gfCNCPoint5[1220] = {X 302.7591, Y 34.0343, Z -6.3333, A 0.000, B 0.000, C 0.000 }
gfCNCPoint5[1221] = {X 293.8549, Y 34.0343, Z -6.3333, A 0.000, B 0.000, C 0.000 }
gfCNCPoint5[1222] = {X 293.8543, Y 40.9020, Z -6.3333, A 0.000, B 0.000, C 0.000 }
gfCNCPoint5[1223] = {X 294.4934, Y 41.5861, Z -6.3333, A 0.000, B 0.000, C 0.000 }
gfCNCPoint5[1224] = {X 294.9740, Y 42.3895, Z -6.3333, A 0.000, B 0.000, C 0.000 }
gfCNCPoint5[1225] = {X 295.2744, Y 43.2762, Z -6.3333, A 0.000, B 0.000, C 0.000 }
gfCNCPoint5[1226] = {X 295.3811, Y 44.2063, Z -6.3333, A 0.000, B 0.000, C 0.000 }
gfCNCPoint5[1227] = {X 295.3811, Y 45.0000, Z -6.3333, A 0.000, B 0.000, C 0.000 }
gfCNCPoint5[1228] = {X 295.2728, Y 45.9613, Z -6.3333, A 0.000, B 0.000, C 0.000 }
gfCNCPoint5[1229] = {X 294.9533, Y 46.8744, Z -6.3333, A 0.000, B 0.000, C 0.000 }
gfCNCPoint5[1230] = {X 294.4386, Y 47.6935, Z -6.3333, A 0.000, B 0.000, C 0.000 }
gfCNCPoint5[1231] = {X 293.7546, Y 48.3775, Z -6.3333, A 0.000, B 0.000, C 0.000 }
gfCNCPoint5[1232] = {X 292.9355, Y 48.8922, Z -6.3333, A 0.000, B 0.000, C 0.000 }
gfCNCPoint5[1233] = {X 292.0224, Y 49.2117, Z -6.3333, A 0.000, B 0.000, C 0.000 }
gfCNCPoint5[1234] = {X 291.0611, Y 49.3200, Z -6.3333, A 0.000, B 0.000, C 0.000 }
gfCNCPoint5[1235] = {X 284.6177, Y 49.3200, Z -6.3333, A 0.000, B 0.000, C 0.000 }
gfCNCPoint5[1236] = {X 283.6613, Y 49.2128, Z -6.3333, A 0.000, B 0.000, C 0.000 }
gfCNCPoint5[1237] = {X 282.7524, Y 48.8965, Z -6.3333, A 0.000, B 0.000, C 0.000 }
gfCNCPoint5[1238] = {X 281.9360, Y 48.3869, Z -6.3333, A 0.000, B 0.000, C 0.000 }
gfCNCPoint5[1239] = {X 281.2527, Y 47.7092, Z -6.3333, A 0.000, B 0.000, C 0.000 }
gfCNCPoint5[1240] = {X 280.7365, Y 46.8970, Z -6.3333, A 0.000, B 0.000, C 0.000 }
gfCNCPoint5[1241] = {X 280.4128, Y 45.9907, Z -6.3333, A 0.000, B 0.000, C 0.000 }
gfCNCPoint5[1242] = {X 280.2978, Y 45.0352, Z -6.3333, A 0.000, B 0.000, C 0.000 }
gfCNCPoint5[1243] = {X 280.2977, Y 44.2074, Z -6.3333, A 0.000, B 0.000, C 0.000 }
gfCNCPoint5[1244] = {X 280.4021, Y 43.2782, Z -6.3333, A 0.000, B 0.000, C 0.000 }
gfCNCPoint5[1245] = {X 280.7020, Y 42.3926, Z -6.3333, A 0.000, B 0.000, C 0.000 }
gfCNCPoint5[1246] = {X 281.1835, Y 41.5911, Z -6.3333, A 0.000, B 0.000, C 0.000 }
gfCNCPoint5[1247] = {X 281.8247, Y 40.9106, Z -6.3333, A 0.000, B 0.000, C 0.000 }
gfCNCPoint5[1248] = {X 281.8245, Y 28.5920, Z -6.3333, A 0.000, B 0.000, C 0.000 }
gfCNCPoint5[1249] = {X 277.8245, Y 28.5921, Z -6.3333, A 0.000, B 0.000, C 0.000 }
gfCNCPoint5[1250] = {X 281.9045, Y 28.5920, Z -6.3333, A 0.000, B 0.000, C 0.000 }
gfCNCPoint5[1251] = {X 281.9043, Y 16.2361, Z -6.3333, A 0.000, B 0.000, C 0.000 }
gfCNCPoint5[1252] = {X 281.2666, Y 15.5757, Z -6.3333, A 0.000, B 0.000, C 0.000 }
gfCNCPoint5[1253] = {X 280.7860, Y 14.7934, Z -6.3333, A 0.000, B 0.000, C 0.000 }
gfCNCPoint5[1254] = {X 280.4850, Y 13.9261, Z -6.3333, A 0.000, B 0.000, C 0.000 }
gfCNCPoint5[1255] = {X 280.3778, Y 13.0143, Z -6.3333, A 0.000, B 0.000, C 0.000 }
gfCNCPoint5[1256] = {X 280.3777, Y 12.1868, Z -6.3333, A 0.000, B 0.000, C 0.000 }
gfCNCPoint5[1257] = {X 280.4840, Y 11.2433, Z -6.3333, A 0.000, B 0.000, C 0.000 }
gfCNCPoint5[1258] = {X 280.7976, Y 10.3472, Z -6.3333, A 0.000, B 0.000, C 0.000 }
gfCNCPoint5[1259] = {X 281.3027, Y 9.5432, Z -6.3333, A 0.000, B 0.000, C 0.000 }
gfCNCPoint5[1260] = {X 281.9741, Y 8.8719, Z -6.3333, A 0.000, B 0.000, C 0.000 }
gfCNCPoint5[1261] = {X 282.7780, Y 8.3667, Z -6.3333, A 0.000, B 0.000, C 0.000 }
gfCNCPoint5[1262] = {X 283.6742, Y 8.0531, Z -6.3333, A 0.000, B 0.000, C 0.000 }
gfCNCPoint5[1263] = {X 284.6177, Y 7.9468, Z -6.3333, A 0.000, B 0.000, C 0.000 }
gfCNCPoint5[1264] = {X 291.0611, Y 7.9468, Z -6.3333, A 0.000, B 0.000, C 0.000 }
gfCNCPoint5[1265] = {X 292.0046, Y 8.0531, Z -6.3333, A 0.000, B 0.000, C 0.000 }
gfCNCPoint5[1266] = {X 292.9008, Y 8.3667, Z -6.3333, A 0.000, B 0.000, C 0.000 }
gfCNCPoint5[1267] = {X 293.7047, Y 8.8718, Z -6.3333, A 0.000, B 0.000, C 0.000 }
gfCNCPoint5[1268] = {X 294.3761, Y 9.5432, Z -6.3333, A 0.000, B 0.000, C 0.000 }
gfCNCPoint5[1269] = {X 294.8812, Y 10.3471, Z -6.3333, A 0.000, B 0.000, C 0.000 }
gfCNCPoint5[1270] = {X 295.1948, Y 11.2433, Z -6.3333, A 0.000, B 0.000, C 0.000 }
gfCNCPoint5[1271] = {X 295.3011, Y 12.1868, Z -6.3333, A 0.000, B 0.000, C 0.000 }
gfCNCPoint5[1272] = {X 295.3011, Y 12.9782, Z -6.3333, A 0.000, B 0.000, C 0.000 }
gfCNCPoint5[1273] = {X 295.1997, Y 13.8997, Z -6.3333, A 0.000, B 0.000, C 0.000 }
gfCNCPoint5[1274] = {X 294.9003, Y 14.7771, Z -6.3333, A 0.000, B 0.000, C 0.000 }
gfCNCPoint5[1275] = {X 294.4175, Y 15.5685, Z -6.3333, A 0.000, B 0.000, C 0.000 }
gfCNCPoint5[1276] = {X 293.7742, Y 16.2360, Z -6.3333, A 0.000, B 0.000, C 0.000 }
gfCNCPoint5[1277] = {X 293.7752, Y 22.2765, Z -6.3333, A 0.000, B 0.000, C 0.000 }
gfCNCPoint5[1278] = {X 302.8386, Y 22.2765, Z -6.3333, A 0.000, B 0.000, C 0.000 }
gfCNCPoint5[1279] = {X 302.8437, Y 16.2401, Z -6.3333, A 0.000, B 0.000, C 0.000 }
gfCNCPoint5[1280] = {X 302.2043, Y 15.5797, Z -6.3333, A 0.000, B 0.000, C 0.000 }
gfCNCPoint5[1281] = {X 301.7222, Y 14.7970, Z -6.3333, A 0.000, B 0.000, C 0.000 }
gfCNCPoint5[1282] = {X 301.4202, Y 13.9287, Z -6.3333, A 0.000, B 0.000, C 0.000 }
gfCNCPoint5[1283] = {X 301.3124, Y 13.0158, Z -6.3333, A 0.000, B 0.000, C 0.000 }
gfCNCPoint5[1284] = {X 301.3123, Y 12.1868, Z -6.3333, A 0.000, B 0.000, C 0.000 }
gfCNCPoint5[1285] = {X 301.4186, Y 11.2433, Z -6.3333, A 0.000, B 0.000, C 0.000 }
gfCNCPoint5[1286] = {X 301.7321, Y 10.3471, Z -6.3333, A 0.000, B 0.000, C 0.000 }
gfCNCPoint5[1287] = {X 302.2373, Y 9.5432, Z -6.3333, A 0.000, B 0.000, C 0.000 }
gfCNCPoint5[1288] = {X 302.9087, Y 8.8718, Z -6.3333, A 0.000, B 0.000, C 0.000 }
gfCNCPoint5[1289] = {X 303.7126, Y 8.3667, Z -6.3333, A 0.000, B 0.000, C 0.000 }
gfCNCPoint5[1290] = {X 304.6088, Y 8.0531, Z -6.3333, A 0.000, B 0.000, C 0.000 }
gfCNCPoint5[1291] = {X 305.5523, Y 7.9468, Z -6.3333, A 0.000, B 0.000, C 0.000 }
gfCNCPoint5[1292] = {X 311.9957, Y 7.9468, Z -6.3333, A 0.000, B 0.000, C 0.000 }
gfCNCPoint5[1293] = {X 312.9392, Y 8.0531, Z -6.3333, A 0.000, B 0.000, C 0.000 }
gfCNCPoint5[1294] = {X 313.8354, Y 8.3667, Z -6.3333, A 0.000, B 0.000, C 0.000 }
gfCNCPoint5[1295] = {X 314.6393, Y 8.8718, Z -6.3333, A 0.000, B 0.000, C 0.000 }
gfCNCPoint5[1296] = {X 315.3107, Y 9.5432, Z -6.3333, A 0.000, B 0.000, C 0.000 }
gfCNCPoint5[1297] = {X 315.8158, Y 10.3471, Z -6.3333, A 0.000, B 0.000, C 0.000 }
gfCNCPoint5[1298] = {X 316.1294, Y 11.2433, Z -6.3333, A 0.000, B 0.000, C 0.000 }
gfCNCPoint5[1299] = {X 316.2357, Y 12.1868, Z -6.3333, A 0.000, B 0.000, C 0.000 }
gfCNCPoint5[1300] = {X 316.2357, Y 12.9782, Z -6.3333, A 0.000, B 0.000, C 0.000 }
gfCNCPoint5[1301] = {X 316.1344, Y 13.8995, Z -6.3333, A 0.000, B 0.000, C 0.000 }
gfCNCPoint5[1302] = {X 315.8352, Y 14.7768, Z -6.3333, A 0.000, B 0.000, C 0.000 }
gfCNCPoint5[1303] = {X 315.3526, Y 15.5682, Z -6.3333, A 0.000, B 0.000, C 0.000 }
gfCNCPoint5[1304] = {X 314.7095, Y 16.2358, Z -6.3333, A 0.000, B 0.000, C 0.000 }
gfCNCPoint5[1305] = {X 314.7087, Y 40.9513, Z -6.3333, A 0.000, B 0.000, C 0.000 }
gfCNCPoint5[1306] = {X 314.7370, Y 40.9741, Z -6.3333, A 0.000, B 0.000, C 0.000 }
gfCNCPoint5[1307] = {X 315.3634, Y 41.6327, Z -6.3333, A 0.000, B 0.000, C 0.000 }
gfCNCPoint5[1308] = {X 315.8351, Y 42.4096, Z -6.3333, A 0.000, B 0.000, C 0.000 }
gfCNCPoint5[1309] = {X 316.1303, Y 43.2692, Z -6.3333, A 0.000, B 0.000, C 0.000 }
gfCNCPoint5[1310] = {X 316.2356, Y 44.1720, Z -6.3333, A 0.000, B 0.000, C 0.000 }
gfCNCPoint5[1311] = {X 316.2357, Y 45.0000, Z -6.3333, A 0.000, B 0.000, C 0.000 }
gfCNCPoint5[1312] = {X 316.1294, Y 45.9435, Z -6.3333, A 0.000, B 0.000, C 0.000 }
gfCNCPoint5[1313] = {X 315.8158, Y 46.8397, Z -6.3333, A 0.000, B 0.000, C 0.000 }
gfCNCPoint5[1314] = {X 315.3107, Y 47.6436, Z -6.3333, A 0.000, B 0.000, C 0.000 }
gfCNCPoint5[1315] = {X 314.6393, Y 48.3150, Z -6.3333, A 0.000, B 0.000, C 0.000 }
gfCNCPoint5[1316] = {X 313.8354, Y 48.8201, Z -6.3333, A 0.000, B 0.000, C 0.000 }
gfCNCPoint5[1317] = {X 312.9392, Y 49.1337, Z -6.3333, A 0.000, B 0.000, C 0.000 }
gfCNCPoint5[1318] = {X 311.9957, Y 49.2400, Z -6.3333, A 0.000, B 0.000, C 0.000 }
gfCNCPoint5[1319] = {X 305.5523, Y 49.2400, Z -6.3333, A 0.000, B 0.000, C 0.000 }
gfCNCPoint5[1320] = {X 304.6135, Y 49.1348, Z -6.3333, A 0.000, B 0.000, C 0.000 }
gfCNCPoint5[1321] = {X 303.7214, Y 48.8243, Z -6.3333, A 0.000, B 0.000, C 0.000 }
gfCNCPoint5[1322] = {X 302.9201, Y 48.3241, Z -6.3333, A 0.000, B 0.000, C 0.000 }
gfCNCPoint5[1323] = {X 302.2495, Y 47.6588, Z -6.3333, A 0.000, B 0.000, C 0.000 }
gfCNCPoint5[1324] = {X 301.7428, Y 46.8616, Z -6.3333, A 0.000, B 0.000, C 0.000 }
gfCNCPoint5[1325] = {X 301.4252, Y 45.9720, Z -6.3333, A 0.000, B 0.000, C 0.000 }
gfCNCPoint5[1326] = {X 301.3124, Y 45.0341, Z -6.3333, A 0.000, B 0.000, C 0.000 }
gfCNCPoint5[1327] = {X 301.3123, Y 44.2032, Z -6.3333, A 0.000, B 0.000, C 0.000 }
gfCNCPoint5[1328] = {X 301.4296, Y 43.2746, Z -6.3333, A 0.000, B 0.000, C 0.000 }
gfCNCPoint5[1329] = {X 301.7327, Y 42.3890, Z -6.3333, A 0.000, B 0.000, C 0.000 }
gfCNCPoint5[1330] = {X 302.2091, Y 41.5833, Z -6.3333, A 0.000, B 0.000, C 0.000 }
gfCNCPoint5[1331] = {X 302.8391, Y 40.8909, Z -6.3333, A 0.000, B 0.000, C 0.000 }
gfCNCPoint5[1332] = {X 302.8391, Y 33.9543, Z -6.3333, A 0.000, B 0.000, C 0.000 }
gfCNCPoint5[1333] = {X 293.7749, Y 33.9543, Z -6.3333, A 0.000, B 0.000, C 0.000 }
gfCNCPoint5[1334] = {X 293.7743, Y 40.9388, Z -6.3333, A 0.000, B 0.000, C 0.000 }
gfCNCPoint5[1335] = {X 294.4130, Y 41.6124, Z -6.3333, A 0.000, B 0.000, C 0.000 }
gfCNCPoint5[1336] = {X 294.8937, Y 42.4065, Z -6.3333, A 0.000, B 0.000, C 0.000 }
gfCNCPoint5[1337] = {X 295.1944, Y 43.2848, Z -6.3333, A 0.000, B 0.000, C 0.000 }
gfCNCPoint5[1338] = {X 295.3011, Y 44.2069, Z -6.3333, A 0.000, B 0.000, C 0.000 }
gfCNCPoint5[1339] = {X 295.3011, Y 45.0000, Z -6.3333, A 0.000, B 0.000, C 0.000 }
gfCNCPoint5[1340] = {X 295.1948, Y 45.9435, Z -6.3333, A 0.000, B 0.000, C 0.000 }
gfCNCPoint5[1341] = {X 294.8812, Y 46.8397, Z -6.3333, A 0.000, B 0.000, C 0.000 }
gfCNCPoint5[1342] = {X 294.3761, Y 47.6436, Z -6.3333, A 0.000, B 0.000, C 0.000 }
gfCNCPoint5[1343] = {X 293.7047, Y 48.3150, Z -6.3333, A 0.000, B 0.000, C 0.000 }
gfCNCPoint5[1344] = {X 292.9008, Y 48.8201, Z -6.3333, A 0.000, B 0.000, C 0.000 }
gfCNCPoint5[1345] = {X 292.0046, Y 49.1337, Z -6.3333, A 0.000, B 0.000, C 0.000 }
gfCNCPoint5[1346] = {X 291.0611, Y 49.2400, Z -6.3333, A 0.000, B 0.000, C 0.000 }
gfCNCPoint5[1347] = {X 284.6177, Y 49.2400, Z -6.3333, A 0.000, B 0.000, C 0.000 }
gfCNCPoint5[1348] = {X 283.6790, Y 49.1348, Z -6.3333, A 0.000, B 0.000, C 0.000 }
gfCNCPoint5[1349] = {X 282.7869, Y 48.8244, Z -6.3333, A 0.000, B 0.000, C 0.000 }
gfCNCPoint5[1350] = {X 281.9857, Y 48.3242, Z -6.3333, A 0.000, B 0.000, C 0.000 }
gfCNCPoint5[1351] = {X 281.3150, Y 47.6590, Z -6.3333, A 0.000, B 0.000, C 0.000 }
gfCNCPoint5[1352] = {X 280.8083, Y 46.8619, Z -6.3333, A 0.000, B 0.000, C 0.000 }
gfCNCPoint5[1353] = {X 280.4907, Y 45.9723, Z -6.3333, A 0.000, B 0.000, C 0.000 }
gfCNCPoint5[1354] = {X 280.3778, Y 45.0345, Z -6.3333, A 0.000, B 0.000, C 0.000 }
gfCNCPoint5[1355] = {X 280.3777, Y 44.2077, Z -6.3333, A 0.000, B 0.000, C 0.000 }
gfCNCPoint5[1356] = {X 280.4822, Y 43.2867, Z -6.3333, A 0.000, B 0.000, C 0.000 }
gfCNCPoint5[1357] = {X 280.7823, Y 42.4096, Z -6.3333, A 0.000, B 0.000, C 0.000 }
gfCNCPoint5[1358] = {X 281.2640, Y 41.6176, Z -6.3333, A 0.000, B 0.000, C 0.000 }
gfCNCPoint5[1359] = {X 281.9047, Y 40.9476, Z -6.3333, A 0.000, B 0.000, C 0.000 }
gfCNCPoint5[1360] = {X 281.9045, Y 28.5920, Z -6.3333, A 0.000, B 0.000, C 0.000 }
gfCNCPoint5[1361] = {X 277.9045, Y 28.5921, Z -6.3333, A 0.000, B 0.000, C 0.000 }
gfCNCPoint5[1362] = {X 281.9845, Y 28.5920, Z -6.3333, A 0.000, B 0.000, C 0.000 }
gfCNCPoint5[1363] = {X 281.9843, Y 16.1984, Z -6.3333, A 0.000, B 0.000, C 0.000 }
gfCNCPoint5[1364] = {X 281.3470, Y 15.5487, Z -6.3333, A 0.000, B 0.000, C 0.000 }
gfCNCPoint5[1365] = {X 280.8663, Y 14.7760, Z -6.3333, A 0.000, B 0.000, C 0.000 }
gfCNCPoint5[1366] = {X 280.5651, Y 13.9173, Z -6.3333, A 0.000, B 0.000, C 0.000 }
gfCNCPoint5[1367] = {X 280.4578, Y 13.0136, Z -6.3333, A 0.000, B 0.000, C 0.000 }
gfCNCPoint5[1368] = {X 280.4577, Y 12.1868, Z -6.3333, A 0.000, B 0.000, C 0.000 }
gfCNCPoint5[1369] = {X 280.5620, Y 11.2611, Z -6.3333, A 0.000, B 0.000, C 0.000 }
gfCNCPoint5[1370] = {X 280.8696, Y 10.3819, Z -6.3333, A 0.000, B 0.000, C 0.000 }
gfCNCPoint5[1371] = {X 281.3652, Y 9.5931, Z -6.3333, A 0.000, B 0.000, C 0.000 }
gfCNCPoint5[1372] = {X 282.0240, Y 8.9344, Z -6.3333, A 0.000, B 0.000, C 0.000 }
gfCNCPoint5[1373] = {X 282.8127, Y 8.4388, Z -6.3333, A 0.000, B 0.000, C 0.000 }
gfCNCPoint5[1374] = {X 283.6920, Y 8.1311, Z -6.3333, A 0.000, B 0.000, C 0.000 }
gfCNCPoint5[1375] = {X 284.6177, Y 8.0268, Z -6.3333, A 0.000, B 0.000, C 0.000 }
gfCNCPoint5[1376] = {X 291.0611, Y 8.0268, Z -6.3333, A 0.000, B 0.000, C 0.000 }
gfCNCPoint5[1377] = {X 291.9868, Y 8.1311, Z -6.3333, A 0.000, B 0.000, C 0.000 }
gfCNCPoint5[1378] = {X 292.8661, Y 8.4388, Z -6.3333, A 0.000, B 0.000, C 0.000 }
gfCNCPoint5[1379] = {X 293.6549, Y 8.9344, Z -6.3333, A 0.000, B 0.000, C 0.000 }
gfCNCPoint5[1380] = {X 294.3136, Y 9.5931, Z -6.3333, A 0.000, B 0.000, C 0.000 }
gfCNCPoint5[1381] = {X 294.8092, Y 10.3819, Z -6.3333, A 0.000, B 0.000, C 0.000 }
gfCNCPoint5[1382] = {X 295.1168, Y 11.2611, Z -6.3333, A 0.000, B 0.000, C 0.000 }
gfCNCPoint5[1383] = {X 295.2211, Y 12.1868, Z -6.3333, A 0.000, B 0.000, C 0.000 }
gfCNCPoint5[1384] = {X 295.2211, Y 12.9782, Z -6.3333, A 0.000, B 0.000, C 0.000 }
gfCNCPoint5[1385] = {X 295.1255, Y 13.8649, Z -6.3333, A 0.000, B 0.000, C 0.000 }
gfCNCPoint5[1386] = {X 294.8430, Y 14.7110, Z -6.3333, A 0.000, B 0.000, C 0.000 }
gfCNCPoint5[1387] = {X 294.3867, Y 15.4773, Z -6.3333, A 0.000, B 0.000, C 0.000 }
gfCNCPoint5[1388] = {X 293.7775, Y 16.1288, Z -6.3333, A 0.000, B 0.000, C 0.000 }
gfCNCPoint5[1389] = {X 293.6942, Y 16.1987, Z -6.3333, A 0.000, B 0.000, C 0.000 }
gfCNCPoint5[1390] = {X 293.6952, Y 22.3565, Z -6.3333, A 0.000, B 0.000, C 0.000 }
gfCNCPoint5[1391] = {X 302.9185, Y 22.3565, Z -6.3333, A 0.000, B 0.000, C 0.000 }
gfCNCPoint5[1392] = {X 302.9237, Y 16.2024, Z -6.3333, A 0.000, B 0.000, C 0.000 }
gfCNCPoint5[1393] = {X 302.2848, Y 15.5527, Z -6.3333, A 0.000, B 0.000, C 0.000 }
gfCNCPoint5[1394] = {X 301.8026, Y 14.7796, Z -6.3333, A 0.000, B 0.000, C 0.000 }
gfCNCPoint5[1395] = {X 301.5003, Y 13.9199, Z -6.3333, A 0.000, B 0.000, C 0.000 }
gfCNCPoint5[1396] = {X 301.3924, Y 13.0151, Z -6.3333, A 0.000, B 0.000, C 0.000 }
gfCNCPoint5[1397] = {X 301.3923, Y 12.1868, Z -6.3333, A 0.000, B 0.000, C 0.000 }
gfCNCPoint5[1398] = {X 301.4966, Y 11.2611, Z -6.3333, A 0.000, B 0.000, C 0.000 }
gfCNCPoint5[1399] = {X 301.8042, Y 10.3819, Z -6.3333, A 0.000, B 0.000, C 0.000 }
gfCNCPoint5[1400] = {X 302.2998, Y 9.5931, Z -6.3333, A 0.000, B 0.000, C 0.000 }
gfCNCPoint5[1401] = {X 302.9585, Y 8.9344, Z -6.3333, A 0.000, B 0.000, C 0.000 }
gfCNCPoint5[1402] = {X 303.7473, Y 8.4388, Z -6.3333, A 0.000, B 0.000, C 0.000 }
gfCNCPoint5[1403] = {X 304.6266, Y 8.1311, Z -6.3333, A 0.000, B 0.000, C 0.000 }
gfCNCPoint5[1404] = {X 305.5523, Y 8.0268, Z -6.3333, A 0.000, B 0.000, C 0.000 }
gfCNCPoint5[1405] = {X 311.9957, Y 8.0268, Z -6.3333, A 0.000, B 0.000, C 0.000 }
gfCNCPoint5[1406] = {X 312.9214, Y 8.1311, Z -6.3333, A 0.000, B 0.000, C 0.000 }
gfCNCPoint5[1407] = {X 313.8007, Y 8.4388, Z -6.3333, A 0.000, B 0.000, C 0.000 }
gfCNCPoint5[1408] = {X 314.5894, Y 8.9344, Z -6.3333, A 0.000, B 0.000, C 0.000 }
gfCNCPoint5[1409] = {X 315.2481, Y 9.5931, Z -6.3333, A 0.000, B 0.000, C 0.000 }
gfCNCPoint5[1410] = {X 315.7438, Y 10.3819, Z -6.3333, A 0.000, B 0.000, C 0.000 }
gfCNCPoint5[1411] = {X 316.0514, Y 11.2611, Z -6.3333, A 0.000, B 0.000, C 0.000 }
gfCNCPoint5[1412] = {X 316.1557, Y 12.1868, Z -6.3333, A 0.000, B 0.000, C 0.000 }
gfCNCPoint5[1413] = {X 316.1557, Y 12.9782, Z -6.3333, A 0.000, B 0.000, C 0.000 }
gfCNCPoint5[1414] = {X 316.0542, Y 13.8913, Z -6.3333, A 0.000, B 0.000, C 0.000 }
gfCNCPoint5[1415] = {X 315.7548, Y 14.7598, Z -6.3333, A 0.000, B 0.000, C 0.000 }
gfCNCPoint5[1416] = {X 315.2721, Y 15.5414, Z -6.3333, A 0.000, B 0.000, C 0.000 }
gfCNCPoint5[1417] = {X 314.6295, Y 16.1981, Z -6.3333, A 0.000, B 0.000, C 0.000 }
gfCNCPoint5[1418] = {X 314.6287, Y 40.9896, Z -6.3333, A 0.000, B 0.000, C 0.000 }
gfCNCPoint5[1419] = {X 314.6838, Y 41.0339, Z -6.3333, A 0.000, B 0.000, C 0.000 }
gfCNCPoint5[1420] = {X 315.2990, Y 41.6801, Z -6.3333, A 0.000, B 0.000, C 0.000 }
gfCNCPoint5[1421] = {X 315.7622, Y 42.4427, Z -6.3333, A 0.000, B 0.000, C 0.000 }
gfCNCPoint5[1422] = {X 316.0522, Y 43.2864, Z -6.3333, A 0.000, B 0.000, C 0.000 }
gfCNCPoint5[1423] = {X 316.1556, Y 44.1727, Z -6.3333, A 0.000, B 0.000, C 0.000 }
gfCNCPoint5[1424] = {X 316.1557, Y 45.0000, Z -6.3333, A 0.000, B 0.000, C 0.000 }
gfCNCPoint5[1425] = {X 316.0514, Y 45.9257, Z -6.3333, A 0.000, B 0.000, C 0.000 }
gfCNCPoint5[1426] = {X 315.7438, Y 46.8050, Z -6.3333, A 0.000, B 0.000, C 0.000 }
gfCNCPoint5[1427] = {X 315.2481, Y 47.5937, Z -6.3333, A 0.000, B 0.000, C 0.000 }
gfCNCPoint5[1428] = {X 314.5894, Y 48.2524, Z -6.3333, A 0.000, B 0.000, C 0.000 }
gfCNCPoint5[1429] = {X 313.8007, Y 48.7480, Z -6.3333, A 0.000, B 0.000, C 0.000 }
gfCNCPoint5[1430] = {X 312.9214, Y 49.0557, Z -6.3333, A 0.000, B 0.000, C 0.000 }
gfCNCPoint5[1431] = {X 311.9957, Y 49.1600, Z -6.3333, A 0.000, B 0.000, C 0.000 }
gfCNCPoint5[1432] = {X 305.5523, Y 49.1600, Z -6.3333, A 0.000, B 0.000, C 0.000 }
gfCNCPoint5[1433] = {X 304.6312, Y 49.0568, Z -6.3333, A 0.000, B 0.000, C 0.000 }
gfCNCPoint5[1434] = {X 303.7559, Y 48.7522, Z -6.3333, A 0.000, B 0.000, C 0.000 }
gfCNCPoint5[1435] = {X 302.9698, Y 48.2613, Z -6.3333, A 0.000, B 0.000, C 0.000 }
gfCNCPoint5[1436] = {X 302.3118, Y 47.6087, Z -6.3333, A 0.000, B 0.000, C 0.000 }
gfCNCPoint5[1437] = {X 301.8147, Y 46.8265, Z -6.3333, A 0.000, B 0.000, C 0.000 }
gfCNCPoint5[1438] = {X 301.5030, Y 45.9537, Z -6.3333, A 0.000, B 0.000, C 0.000 }
gfCNCPoint5[1439] = {X 301.3924, Y 45.0335, Z -6.3333, A 0.000, B 0.000, C 0.000 }
gfCNCPoint5[1440] = {X 301.3923, Y 44.2051, Z -6.3333, A 0.000, B 0.000, C 0.000 }
gfCNCPoint5[1441] = {X 301.5095, Y 43.2839, Z -6.3333, A 0.000, B 0.000, C 0.000 }
gfCNCPoint5[1442] = {X 301.8128, Y 42.4063, Z -6.3333, A 0.000, B 0.000, C 0.000 }
gfCNCPoint5[1443] = {X 302.2894, Y 41.6093, Z -6.3333, A 0.000, B 0.000, C 0.000 }
gfCNCPoint5[1444] = {X 302.9191, Y 40.9268, Z -6.3333, A 0.000, B 0.000, C 0.000 }
gfCNCPoint5[1445] = {X 302.9191, Y 33.8743, Z -6.3333, A 0.000, B 0.000, C 0.000 }
gfCNCPoint5[1446] = {X 293.6950, Y 33.8743, Z -6.3333, A 0.000, B 0.000, C 0.000 }
gfCNCPoint5[1447] = {X 293.6943, Y 40.9760, Z -6.3333, A 0.000, B 0.000, C 0.000 }
gfCNCPoint5[1448] = {X 294.3326, Y 41.6390, Z -6.3333, A 0.000, B 0.000, C 0.000 }
gfCNCPoint5[1449] = {X 294.8134, Y 42.4237, Z -6.3333, A 0.000, B 0.000, C 0.000 }
gfCNCPoint5[1450] = {X 295.1143, Y 43.2935, Z -6.3333, A 0.000, B 0.000, C 0.000 }
gfCNCPoint5[1451] = {X 295.2211, Y 44.2076, Z -6.3333, A 0.000, B 0.000, C 0.000 }
gfCNCPoint5[1452] = {X 295.2211, Y 45.0000, Z -6.3333, A 0.000, B 0.000, C 0.000 }
gfCNCPoint5[1453] = {X 295.1168, Y 45.9257, Z -6.3333, A 0.000, B 0.000, C 0.000 }
gfCNCPoint5[1454] = {X 294.8092, Y 46.8050, Z -6.3333, A 0.000, B 0.000, C 0.000 }
gfCNCPoint5[1455] = {X 294.3136, Y 47.5937, Z -6.3333, A 0.000, B 0.000, C 0.000 }
gfCNCPoint5[1456] = {X 293.6549, Y 48.2524, Z -6.3333, A 0.000, B 0.000, C 0.000 }
gfCNCPoint5[1457] = {X 292.8661, Y 48.7480, Z -6.3333, A 0.000, B 0.000, C 0.000 }
gfCNCPoint5[1458] = {X 291.9868, Y 49.0557, Z -6.3333, A 0.000, B 0.000, C 0.000 }
gfCNCPoint5[1459] = {X 291.0611, Y 49.1600, Z -6.3333, A 0.000, B 0.000, C 0.000 }
gfCNCPoint5[1460] = {X 284.6177, Y 49.1600, Z -6.3333, A 0.000, B 0.000, C 0.000 }
gfCNCPoint5[1461] = {X 283.6967, Y 49.0568, Z -6.3333, A 0.000, B 0.000, C 0.000 }
gfCNCPoint5[1462] = {X 282.8214, Y 48.7522, Z -6.3333, A 0.000, B 0.000, C 0.000 }
gfCNCPoint5[1463] = {X 282.0353, Y 48.2615, Z -6.3333, A 0.000, B 0.000, C 0.000 }
gfCNCPoint5[1464] = {X 281.3774, Y 47.6088, Z -6.3333, A 0.000, B 0.000, C 0.000 }
gfCNCPoint5[1465] = {X 280.8802, Y 46.8267, Z -6.3333, A 0.000, B 0.000, C 0.000 }
gfCNCPoint5[1466] = {X 280.5685, Y 45.9540, Z -6.3333, A 0.000, B 0.000, C 0.000 }
gfCNCPoint5[1467] = {X 280.4578, Y 45.0339, Z -6.3333, A 0.000, B 0.000, C 0.000 }
gfCNCPoint5[1468] = {X 280.4577, Y 44.2081, Z -6.3333, A 0.000, B 0.000, C 0.000 }
gfCNCPoint5[1469] = {X 280.5623, Y 43.2952, Z -6.3333, A 0.000, B 0.000, C 0.000 }
gfCNCPoint5[1470] = {X 280.8627, Y 42.4267, Z -6.3333, A 0.000, B 0.000, C 0.000 }
gfCNCPoint5[1471] = {X 281.3445, Y 41.6443, Z -6.3333, A 0.000, B 0.000, C 0.000 }
gfCNCPoint5[1472] = {X 281.9847, Y 40.9851, Z -6.3333, A 0.000, B 0.000, C 0.000 }
gfCNCPoint5[1473] = {X 281.9845, Y 28.5920, Z -6.3333, A 0.000, B 0.000, C 0.000 }
gfCNCPoint5[1474] = {X 277.9845, Y 28.5921, Z -6.3333, A 0.000, B 0.000, C 0.000 }
gfCNCPoint5[1475] = {X 282.0645, Y 28.5920, Z -6.3333, A 0.000, B 0.000, C 0.000 }
gfCNCPoint5[1476] = {X 282.0643, Y 16.1603, Z -6.3333, A 0.000, B 0.000, C 0.000 }
gfCNCPoint5[1477] = {X 281.4275, Y 15.5215, Z -6.3333, A 0.000, B 0.000, C 0.000 }
gfCNCPoint5[1478] = {X 280.9467, Y 14.7585, Z -6.3333, A 0.000, B 0.000, C 0.000 }
gfCNCPoint5[1479] = {X 280.6452, Y 13.9084, Z -6.3333, A 0.000, B 0.000, C 0.000 }
gfCNCPoint5[1480] = {X 280.5378, Y 13.0129, Z -6.3333, A 0.000, B 0.000, C 0.000 }
gfCNCPoint5[1481] = {X 280.5377, Y 12.1868, Z -6.3333, A 0.000, B 0.000, C 0.000 }
gfCNCPoint5[1482] = {X 280.6400, Y 11.2789, Z -6.3333, A 0.000, B 0.000, C 0.000 }
gfCNCPoint5[1483] = {X 280.9417, Y 10.4166, Z -6.3333, A 0.000, B 0.000, C 0.000 }
gfCNCPoint5[1484] = {X 281.4278, Y 9.6430, Z -6.3333, A 0.000, B 0.000, C 0.000 }
gfCNCPoint5[1485] = {X 282.0738, Y 8.9969, Z -6.3333, A 0.000, B 0.000, C 0.000 }
gfCNCPoint5[1486] = {X 282.8474, Y 8.5109, Z -6.3333, A 0.000, B 0.000, C 0.000 }
gfCNCPoint5[1487] = {X 283.7098, Y 8.2091, Z -6.3333, A 0.000, B 0.000, C 0.000 }
gfCNCPoint5[1488] = {X 284.6177, Y 8.1068, Z -6.3333, A 0.000, B 0.000, C 0.000 }
gfCNCPoint5[1489] = {X 291.0611, Y 8.1068, Z -6.3333, A 0.000, B 0.000, C 0.000 }
gfCNCPoint5[1490] = {X 291.9690, Y 8.2091, Z -6.3333, A 0.000, B 0.000, C 0.000 }
gfCNCPoint5[1491] = {X 292.8314, Y 8.5109, Z -6.3333, A 0.000, B 0.000, C 0.000 }
gfCNCPoint5[1492] = {X 293.6050, Y 8.9969, Z -6.3333, A 0.000, B 0.000, C 0.000 }
gfCNCPoint5[1493] = {X 294.2510, Y 9.6430, Z -6.3333, A 0.000, B 0.000, C 0.000 }
gfCNCPoint5[1494] = {X 294.7371, Y 10.4166, Z -6.3333, A 0.000, B 0.000, C 0.000 }
gfCNCPoint5[1495] = {X 295.0388, Y 11.2789, Z -6.3333, A 0.000, B 0.000, C 0.000 }
gfCNCPoint5[1496] = {X 295.1411, Y 12.1868, Z -6.3333, A 0.000, B 0.000, C 0.000 }
gfCNCPoint5[1497] = {X 295.1411, Y 12.9782, Z -6.3333, A 0.000, B 0.000, C 0.000 }
gfCNCPoint5[1498] = {X 295.0473, Y 13.8479, Z -6.3333, A 0.000, B 0.000, C 0.000 }
gfCNCPoint5[1499] = {X 294.7703, Y 14.6776, Z -6.3333, A 0.000, B 0.000, C 0.000 }
gfCNCPoint5[1500] = {X 294.3227, Y 15.4292, Z -6.3333, A 0.000, B 0.000, C 0.000 }
gfCNCPoint5[1501] = {X 293.7252, Y 16.0682, Z -6.3333, A 0.000, B 0.000, C 0.000 }
gfCNCPoint5[1502] = {X 293.6677, Y 16.1168, Z -6.3333, A 0.000, B 0.000, C 0.000 }
gfCNCPoint5[1503] = {X 293.6093, Y 16.1644, Z -6.3333, A 0.000, B 0.000, C 0.000 }
gfCNCPoint5[1504] = {X 293.6142, Y 16.1987, Z -6.3333, A 0.000, B 0.000, C 0.000 }
gfCNCPoint5[1505] = {X 293.6152, Y 22.4365, Z -6.3333, A 0.000, B 0.000, C 0.000 }
gfCNCPoint5[1506] = {X 302.9985, Y 22.4365, Z -6.3333, A 0.000, B 0.000, C 0.000 }
gfCNCPoint5[1507] = {X 303.0038, Y 16.1642, Z -6.3333, A 0.000, B 0.000, C 0.000 }
gfCNCPoint5[1508] = {X 302.9453, Y 16.1166, Z -6.3333, A 0.000, B 0.000, C 0.000 }
gfCNCPoint5[1509] = {X 302.8878, Y 16.0678, Z -6.3333, A 0.000, B 0.000, C 0.000 }
gfCNCPoint5[1510] = {X 302.2959, Y 15.4362, Z -6.3333, A 0.000, B 0.000, C 0.000 }
gfCNCPoint5[1511] = {X 301.8506, Y 14.6939, Z -6.3333, A 0.000, B 0.000, C 0.000 }
gfCNCPoint5[1512] = {X 301.5719, Y 13.8743, Z -6.3333, A 0.000, B 0.000, C 0.000 }
gfCNCPoint5[1513] = {X 301.4724, Y 13.0144, Z -6.3333, A 0.000, B 0.000, C 0.000 }
gfCNCPoint5[1514] = {X 301.4723, Y 12.1868, Z -6.3333, A 0.000, B 0.000, C 0.000 }
gfCNCPoint5[1515] = {X 301.5745, Y 11.2789, Z -6.3333, A 0.000, B 0.000, C 0.000 }
gfCNCPoint5[1516] = {X 301.8763, Y 10.4166, Z -6.3333, A 0.000, B 0.000, C 0.000 }
gfCNCPoint5[1517] = {X 302.3624, Y 9.6430, Z -6.3333, A 0.000, B 0.000, C 0.000 }
gfCNCPoint5[1518] = {X 303.0084, Y 8.9969, Z -6.3333, A 0.000, B 0.000, C 0.000 }
gfCNCPoint5[1519] = {X 303.7820, Y 8.5109, Z -6.3333, A 0.000, B 0.000, C 0.000 }
gfCNCPoint5[1520] = {X 304.6444, Y 8.2091, Z -6.3333, A 0.000, B 0.000, C 0.000 }
gfCNCPoint5[1521] = {X 305.5523, Y 8.1068, Z -6.3333, A 0.000, B 0.000, C 0.000 }
gfCNCPoint5[1522] = {X 311.9957, Y 8.1068, Z -6.3333, A 0.000, B 0.000, C 0.000 }
gfCNCPoint5[1523] = {X 312.9036, Y 8.2091, Z -6.3333, A 0.000, B 0.000, C 0.000 }
gfCNCPoint5[1524] = {X 313.7660, Y 8.5109, Z -6.3333, A 0.000, B 0.000, C 0.000 }
gfCNCPoint5[1525] = {X 314.5396, Y 8.9969, Z -6.3333, A 0.000, B 0.000, C 0.000 }
gfCNCPoint5[1526] = {X 315.1856, Y 9.6430, Z -6.3333, A 0.000, B 0.000, C 0.000 }
gfCNCPoint5[1527] = {X 315.6717, Y 10.4166, Z -6.3333, A 0.000, B 0.000, C 0.000 }
gfCNCPoint5[1528] = {X 315.9734, Y 11.2789, Z -6.3333, A 0.000, B 0.000, C 0.000 }
gfCNCPoint5[1529] = {X 316.0757, Y 12.1868, Z -6.3333, A 0.000, B 0.000, C 0.000 }
gfCNCPoint5[1530] = {X 316.0757, Y 12.9782, Z -6.3333, A 0.000, B 0.000, C 0.000 }
gfCNCPoint5[1531] = {X 315.9741, Y 13.8829, Z -6.3333, A 0.000, B 0.000, C 0.000 }
gfCNCPoint5[1532] = {X 315.6744, Y 14.7426, Z -6.3333, A 0.000, B 0.000, C 0.000 }
gfCNCPoint5[1533] = {X 315.1915, Y 15.5144, Z -6.3333, A 0.000, B 0.000, C 0.000 }
gfCNCPoint5[1534] = {X 314.5495, Y 16.1599, Z -6.3333, A 0.000, B 0.000, C 0.000 }
gfCNCPoint5[1535] = {X 314.5487, Y 41.0279, Z -6.3333, A 0.000, B 0.000, C 0.000 }
gfCNCPoint5[1536] = {X 314.6336, Y 41.0962, Z -6.3333, A 0.000, B 0.000, C 0.000 }
gfCNCPoint5[1537] = {X 315.2363, Y 41.7299, Z -6.3333, A 0.000, B 0.000, C 0.000 }
gfCNCPoint5[1538] = {X 315.6902, Y 42.4775, Z -6.3333, A 0.000, B 0.000, C 0.000 }
gfCNCPoint5[1539] = {X 315.9743, Y 43.3047, Z -6.3333, A 0.000, B 0.000, C 0.000 }
gfCNCPoint5[1540] = {X 316.0756, Y 44.1734, Z -6.3333, A 0.000, B 0.000, C 0.000 }
gfCNCPoint5[1541] = {X 316.0757, Y 45.0000, Z -6.3333, A 0.000, B 0.000, C 0.000 }
gfCNCPoint5[1542] = {X 315.9734, Y 45.9079, Z -6.3333, A 0.000, B 0.000, C 0.000 }
gfCNCPoint5[1543] = {X 315.6717, Y 46.7702, Z -6.3333, A 0.000, B 0.000, C 0.000 }
gfCNCPoint5[1544] = {X 315.1856, Y 47.5438, Z -6.3333, A 0.000, B 0.000, C 0.000 }
gfCNCPoint5[1545] = {X 314.5396, Y 48.1899, Z -6.3333, A 0.000, B 0.000, C 0.000 }
gfCNCPoint5[1546] = {X 313.7660, Y 48.6760, Z -6.3333, A 0.000, B 0.000, C 0.000 }
gfCNCPoint5[1547] = {X 312.9036, Y 48.9777, Z -6.3333, A 0.000, B 0.000, C 0.000 }
gfCNCPoint5[1548] = {X 311.9957, Y 49.0800, Z -6.3333, A 0.000, B 0.000, C 0.000 }
gfCNCPoint5[1549] = {X 305.5523, Y 49.0800, Z -6.3333, A 0.000, B 0.000, C 0.000 }
gfCNCPoint5[1550] = {X 304.6489, Y 48.9787, Z -6.3333, A 0.000, B 0.000, C 0.000 }
gfCNCPoint5[1551] = {X 303.7905, Y 48.6800, Z -6.3333, A 0.000, B 0.000, C 0.000 }
gfCNCPoint5[1552] = {X 303.0194, Y 48.1986, Z -6.3333, A 0.000, B 0.000, C 0.000 }
gfCNCPoint5[1553] = {X 302.3741, Y 47.5585, Z -6.3333, A 0.000, B 0.000, C 0.000 }
gfCNCPoint5[1554] = {X 301.8865, Y 46.7914, Z -6.3333, A 0.000, B 0.000, C 0.000 }
gfCNCPoint5[1555] = {X 301.5809, Y 45.9353, Z -6.3333, A 0.000, B 0.000, C 0.000 }
gfCNCPoint5[1556] = {X 301.4724, Y 45.0328, Z -6.3333, A 0.000, B 0.000, C 0.000 }
gfCNCPoint5[1557] = {X 301.4723, Y 44.2070, Z -6.3333, A 0.000, B 0.000, C 0.000 }
gfCNCPoint5[1558] = {X 301.5895, Y 43.2934, Z -6.3333, A 0.000, B 0.000, C 0.000 }
gfCNCPoint5[1559] = {X 301.8930, Y 42.4238, Z -6.3333, A 0.000, B 0.000, C 0.000 }
gfCNCPoint5[1560] = {X 302.3697, Y 41.6357, Z -6.3333, A 0.000, B 0.000, C 0.000 }
gfCNCPoint5[1561] = {X 302.9991, Y 40.9632, Z -6.3333, A 0.000, B 0.000, C 0.000 }
gfCNCPoint5[1562] = {X 302.9991, Y 33.7943, Z -6.3333, A 0.000, B 0.000, C 0.000 }
gfCNCPoint5[1563] = {X 293.6150, Y 33.7943, Z -6.3333, A 0.000, B 0.000, C 0.000 }
gfCNCPoint5[1564] = {X 293.6143, Y 41.0136, Z -6.3333, A 0.000, B 0.000, C 0.000 }
gfCNCPoint5[1565] = {X 294.2521, Y 41.6659, Z -6.3333, A 0.000, B 0.000, C 0.000 }
gfCNCPoint5[1566] = {X 294.7331, Y 42.4411, Z -6.3333, A 0.000, B 0.000, C 0.000 }
gfCNCPoint5[1567] = {X 295.0342, Y 43.3022, Z -6.3333, A 0.000, B 0.000, C 0.000 }
gfCNCPoint5[1568] = {X 295.1411, Y 44.2082, Z -6.3333, A 0.000, B 0.000, C 0.000 }
gfCNCPoint5[1569] = {X 295.1411, Y 45.0000, Z -6.3333, A 0.000, B 0.000, C 0.000 }
gfCNCPoint5[1570] = {X 295.0388, Y 45.9079, Z -6.3333, A 0.000, B 0.000, C 0.000 }
gfCNCPoint5[1571] = {X 294.7371, Y 46.7702, Z -6.3333, A 0.000, B 0.000, C 0.000 }
gfCNCPoint5[1572] = {X 294.2510, Y 47.5438, Z -6.3333, A 0.000, B 0.000, C 0.000 }
gfCNCPoint5[1573] = {X 293.6050, Y 48.1899, Z -6.3333, A 0.000, B 0.000, C 0.000 }
gfCNCPoint5[1574] = {X 292.8314, Y 48.6760, Z -6.3333, A 0.000, B 0.000, C 0.000 }
gfCNCPoint5[1575] = {X 291.9690, Y 48.9777, Z -6.3333, A 0.000, B 0.000, C 0.000 }
gfCNCPoint5[1576] = {X 291.0611, Y 49.0800, Z -6.3333, A 0.000, B 0.000, C 0.000 }
gfCNCPoint5[1577] = {X 284.6177, Y 49.0800, Z -6.3333, A 0.000, B 0.000, C 0.000 }
gfCNCPoint5[1578] = {X 283.7144, Y 48.9788, Z -6.3333, A 0.000, B 0.000, C 0.000 }
gfCNCPoint5[1579] = {X 282.8560, Y 48.6801, Z -6.3333, A 0.000, B 0.000, C 0.000 }
gfCNCPoint5[1580] = {X 282.0850, Y 48.1987, Z -6.3333, A 0.000, B 0.000, C 0.000 }
gfCNCPoint5[1581] = {X 281.4397, Y 47.5587, Z -6.3333, A 0.000, B 0.000, C 0.000 }
gfCNCPoint5[1582] = {X 280.9521, Y 46.7916, Z -6.3333, A 0.000, B 0.000, C 0.000 }
gfCNCPoint5[1583] = {X 280.6464, Y 45.9356, Z -6.3333, A 0.000, B 0.000, C 0.000 }
gfCNCPoint5[1584] = {X 280.5378, Y 45.0332, Z -6.3333, A 0.000, B 0.000, C 0.000 }
gfCNCPoint5[1585] = {X 280.5377, Y 44.2085, Z -6.3333, A 0.000, B 0.000, C 0.000 }
gfCNCPoint5[1586] = {X 280.6424, Y 43.3038, Z -6.3333, A 0.000, B 0.000, C 0.000 }
gfCNCPoint5[1587] = {X 280.9430, Y 42.4440, Z -6.3333, A 0.000, B 0.000, C 0.000 }
gfCNCPoint5[1588] = {X 281.4250, Y 41.6712, Z -6.3333, A 0.000, B 0.000, C 0.000 }
gfCNCPoint5[1589] = {X 282.0647, Y 41.0230, Z -6.3333, A 0.000, B 0.000, C 0.000 }
gfCNCPoint5[1590] = {X 282.0645, Y 28.5920, Z -6.3333, A 0.000, B 0.000, C 0.000 }
gfCNCPoint5[1591] = {X 278.0645, Y 28.5921, Z -6.3333, A 0.000, B 0.000, C 0.000 }
gfCNCPoint5[1592] = {X 282.1445, Y 28.5920, Z -6.3333, A 0.000, B 0.000, C 0.000 }
gfCNCPoint5[1593] = {X 282.1443, Y 16.1217, Z -6.3333, A 0.000, B 0.000, C 0.000 }
gfCNCPoint5[1594] = {X 281.5027, Y 15.4873, Z -6.3333, A 0.000, B 0.000, C 0.000 }
gfCNCPoint5[1595] = {X 281.0195, Y 14.7254, Z -6.3333, A 0.000, B 0.000, C 0.000 }
gfCNCPoint5[1596] = {X 280.7194, Y 13.8745, Z -6.3333, A 0.000, B 0.000, C 0.000 }
gfCNCPoint5[1597] = {X 280.6177, Y 12.9780, Z -6.3333, A 0.000, B 0.000, C 0.000 }
gfCNCPoint5[1598] = {X 280.6177, Y 12.1868, Z -6.3333, A 0.000, B 0.000, C 0.000 }
gfCNCPoint5[1599] = {X 280.7180, Y 11.2967, Z -6.3333, A 0.000, B 0.000, C 0.000 }
gfCNCPoint5[1600] = {X 281.0138, Y 10.4513, Z -6.3333, A 0.000, B 0.000, C 0.000 }
gfCNCPoint5[1601] = {X 281.4903, Y 9.6929, Z -6.3333, A 0.000, B 0.000, C 0.000 }
gfCNCPoint5[1602] = {X 282.1237, Y 9.0595, Z -6.3333, A 0.000, B 0.000, C 0.000 }
gfCNCPoint5[1603] = {X 282.8821, Y 8.5829, Z -6.3333, A 0.000, B 0.000, C 0.000 }
gfCNCPoint5[1604] = {X 283.7276, Y 8.2871, Z -6.3333, A 0.000, B 0.000, C 0.000 }
gfCNCPoint5[1605] = {X 284.6177, Y 8.1868, Z -6.3333, A 0.000, B 0.000, C 0.000 }
gfCNCPoint5[1606] = {X 291.0611, Y 8.1868, Z -6.3333, A 0.000, B 0.000, C 0.000 }
gfCNCPoint5[1607] = {X 291.9512, Y 8.2871, Z -6.3333, A 0.000, B 0.000, C 0.000 }
gfCNCPoint5[1608] = {X 292.7967, Y 8.5829, Z -6.3333, A 0.000, B 0.000, C 0.000 }
gfCNCPoint5[1609] = {X 293.5551, Y 9.0595, Z -6.3333, A 0.000, B 0.000, C 0.000 }
gfCNCPoint5[1610] = {X 294.1885, Y 9.6929, Z -6.3333, A 0.000, B 0.000, C 0.000 }
gfCNCPoint5[1611] = {X 294.6650, Y 10.4513, Z -6.3333, A 0.000, B 0.000, C 0.000 }
gfCNCPoint5[1612] = {X 294.9608, Y 11.2967, Z -6.3333, A 0.000, B 0.000, C 0.000 }
gfCNCPoint5[1613] = {X 295.0611, Y 12.1868, Z -6.3333, A 0.000, B 0.000, C 0.000 }
gfCNCPoint5[1614] = {X 295.0609, Y 13.0192, Z -6.3333, A 0.000, B 0.000, C 0.000 }
gfCNCPoint5[1615] = {X 294.9625, Y 13.8609, Z -6.3333, A 0.000, B 0.000, C 0.000 }
gfCNCPoint5[1616] = {X 294.6890, Y 14.6629, Z -6.3333, A 0.000, B 0.000, C 0.000 }
gfCNCPoint5[1617] = {X 294.2526, Y 15.3894, Z -6.3333, A 0.000, B 0.000, C 0.000 }
gfCNCPoint5[1618] = {X 293.6730, Y 16.0076, Z -6.3333, A 0.000, B 0.000, C 0.000 }
gfCNCPoint5[1619] = {X 293.5961, Y 16.0722, Z -6.3333, A 0.000, B 0.000, C 0.000 }
gfCNCPoint5[1620] = {X 293.5177, Y 16.1348, Z -6.3333, A 0.000, B 0.000, C 0.000 }
gfCNCPoint5[1621] = {X 293.5342, Y 16.1926, Z -6.3333, A 0.000, B 0.000, C 0.000 }
gfCNCPoint5[1622] = {X 293.5352, Y 22.5165, Z -6.3333, A 0.000, B 0.000, C 0.000 }
gfCNCPoint5[1623] = {X 302.6785, Y 22.5165, Z -6.3333, A 0.000, B 0.000, C 0.000 }
gfCNCPoint5[1624] = {X 303.0785, Y 22.5166, Z -6.3333, A 0.000, B 0.000, C 0.000 }
gfCNCPoint5[1625] = {X 303.0788, Y 16.1927, Z -6.3333, A 0.000, B 0.000, C 0.000 }
gfCNCPoint5[1626] = {X 303.0955, Y 16.1346, Z -6.3333, A 0.000, B 0.000, C 0.000 }
gfCNCPoint5[1627] = {X 303.0170, Y 16.0719, Z -6.3333, A 0.000, B 0.000, C 0.000 }
gfCNCPoint5[1628] = {X 302.9400, Y 16.0073, Z -6.3333, A 0.000, B 0.000, C 0.000 }
gfCNCPoint5[1629] = {X 302.3544, Y 15.3808, Z -6.3333, A 0.000, B 0.000, C 0.000 }
gfCNCPoint5[1630] = {X 301.9157, Y 14.6440, Z -6.3333, A 0.000, B 0.000, C 0.000 }
gfCNCPoint5[1631] = {X 301.6442, Y 13.8306, Z -6.3333, A 0.000, B 0.000, C 0.000 }
gfCNCPoint5[1632] = {X 301.5523, Y 12.9780, Z -6.3333, A 0.000, B 0.000, C 0.000 }
gfCNCPoint5[1633] = {X 301.5523, Y 12.1868, Z -6.3333, A 0.000, B 0.000, C 0.000 }
gfCNCPoint5[1634] = {X 301.6525, Y 11.2967, Z -6.3333, A 0.000, B 0.000, C 0.000 }
gfCNCPoint5[1635] = {X 301.9484, Y 10.4513, Z -6.3333, A 0.000, B 0.000, C 0.000 }
gfCNCPoint5[1636] = {X 302.4249, Y 9.6929, Z -6.3333, A 0.000, B 0.000, C 0.000 }
gfCNCPoint5[1637] = {X 303.0583, Y 9.0595, Z -6.3333, A 0.000, B 0.000, C 0.000 }
gfCNCPoint5[1638] = {X 303.8167, Y 8.5829, Z -6.3333, A 0.000, B 0.000, C 0.000 }
gfCNCPoint5[1639] = {X 304.6622, Y 8.2871, Z -6.3333, A 0.000, B 0.000, C 0.000 }
gfCNCPoint5[1640] = {X 305.5523, Y 8.1868, Z -6.3333, A 0.000, B 0.000, C 0.000 }
gfCNCPoint5[1641] = {X 311.9957, Y 8.1868, Z -6.3333, A 0.000, B 0.000, C 0.000 }
gfCNCPoint5[1642] = {X 312.8858, Y 8.2871, Z -6.3333, A 0.000, B 0.000, C 0.000 }
gfCNCPoint5[1643] = {X 313.7313, Y 8.5829, Z -6.3333, A 0.000, B 0.000, C 0.000 }
gfCNCPoint5[1644] = {X 314.4897, Y 9.0595, Z -6.3333, A 0.000, B 0.000, C 0.000 }
gfCNCPoint5[1645] = {X 315.1230, Y 9.6929, Z -6.3333, A 0.000, B 0.000, C 0.000 }
gfCNCPoint5[1646] = {X 315.5996, Y 10.4513, Z -6.3333, A 0.000, B 0.000, C 0.000 }
gfCNCPoint5[1647] = {X 315.8954, Y 11.2967, Z -6.3333, A 0.000, B 0.000, C 0.000 }
gfCNCPoint5[1648] = {X 315.9957, Y 12.1868, Z -6.3333, A 0.000, B 0.000, C 0.000 }
gfCNCPoint5[1649] = {X 315.9955, Y 13.0192, Z -6.3333, A 0.000, B 0.000, C 0.000 }
gfCNCPoint5[1650] = {X 315.8870, Y 13.9044, Z -6.3333, A 0.000, B 0.000, C 0.000 }
gfCNCPoint5[1651] = {X 315.5850, Y 14.7436, Z -6.3333, A 0.000, B 0.000, C 0.000 }
gfCNCPoint5[1652] = {X 315.1045, Y 15.4950, Z -6.3333, A 0.000, B 0.000, C 0.000 }
gfCNCPoint5[1653] = {X 314.4695, Y 16.1213, Z -6.3333, A 0.000, B 0.000, C 0.000 }
gfCNCPoint5[1654] = {X 314.4687, Y 41.0661, Z -6.3333, A 0.000, B 0.000, C 0.000 }
gfCNCPoint5[1655] = {X 314.6075, Y 41.1792, Z -6.3333, A 0.000, B 0.000, C 0.000 }
gfCNCPoint5[1656] = {X 315.1934, Y 41.8056, Z -6.3333, A 0.000, B 0.000, C 0.000 }
gfCNCPoint5[1657] = {X 315.6322, Y 42.5426, Z -6.3333, A 0.000, B 0.000, C 0.000 }
gfCNCPoint5[1658] = {X 315.9038, Y 43.3561, Z -6.3333, A 0.000, B 0.000, C 0.000 }
gfCNCPoint5[1659] = {X 315.9957, Y 44.2089, Z -6.3333, A 0.000, B 0.000, C 0.000 }
gfCNCPoint5[1660] = {X 315.9957, Y 45.0000, Z -6.3333, A 0.000, B 0.000, C 0.000 }
gfCNCPoint5[1661] = {X 315.8954, Y 45.8901, Z -6.3333, A 0.000, B 0.000, C 0.000 }
gfCNCPoint5[1662] = {X 315.5996, Y 46.7355, Z -6.3333, A 0.000, B 0.000, C 0.000 }
gfCNCPoint5[1663] = {X 315.1230, Y 47.4940, Z -6.3333, A 0.000, B 0.000, C 0.000 }
gfCNCPoint5[1664] = {X 314.4897, Y 48.1273, Z -6.3333, A 0.000, B 0.000, C 0.000 }
gfCNCPoint5[1665] = {X 313.7313, Y 48.6039, Z -6.3333, A 0.000, B 0.000, C 0.000 }
gfCNCPoint5[1666] = {X 312.8858, Y 48.8997, Z -6.3333, A 0.000, B 0.000, C 0.000 }
gfCNCPoint5[1667] = {X 311.9957, Y 49.0000, Z -6.3333, A 0.000, B 0.000, C 0.000 }
gfCNCPoint5[1668] = {X 305.5523, Y 49.0000, Z -6.3333, A 0.000, B 0.000, C 0.000 }
gfCNCPoint5[1669] = {X 304.6622, Y 48.8997, Z -6.3333, A 0.000, B 0.000, C 0.000 }
gfCNCPoint5[1670] = {X 303.8167, Y 48.6039, Z -6.3333, A 0.000, B 0.000, C 0.000 }
gfCNCPoint5[1671] = {X 303.0583, Y 48.1273, Z -6.3333, A 0.000, B 0.000, C 0.000 }
gfCNCPoint5[1672] = {X 302.4249, Y 47.4939, Z -6.3333, A 0.000, B 0.000, C 0.000 }
gfCNCPoint5[1673] = {X 301.9484, Y 46.7355, Z -6.3333, A 0.000, B 0.000, C 0.000 }
gfCNCPoint5[1674] = {X 301.6525, Y 45.8901, Z -6.3333, A 0.000, B 0.000, C 0.000 }
gfCNCPoint5[1675] = {X 301.5523, Y 45.0000, Z -6.3333, A 0.000, B 0.000, C 0.000 }
gfCNCPoint5[1676] = {X 301.5523, Y 44.2089, Z -6.3333, A 0.000, B 0.000, C 0.000 }
gfCNCPoint5[1677] = {X 301.6694, Y 43.3029, Z -6.3333, A 0.000, B 0.000, C 0.000 }
gfCNCPoint5[1678] = {X 301.9732, Y 42.4414, Z -6.3333, A 0.000, B 0.000, C 0.000 }
gfCNCPoint5[1679] = {X 302.4500, Y 41.6623, Z -6.3333, A 0.000, B 0.000, C 0.000 }
gfCNCPoint5[1680] = {X 303.0791, Y 40.9999, Z -6.3333, A 0.000, B 0.000, C 0.000 }
gfCNCPoint5[1681] = {X 303.0791, Y 33.7143, Z -6.3333, A 0.000, B 0.000, C 0.000 }
gfCNCPoint5[1682] = {X 293.5350, Y 33.7143, Z -6.3333, A 0.000, B 0.000, C 0.000 }
gfCNCPoint5[1683] = {X 293.5343, Y 41.0517, Z -6.3333, A 0.000, B 0.000, C 0.000 }
gfCNCPoint5[1684] = {X 294.1716, Y 41.6930, Z -6.3333, A 0.000, B 0.000, C 0.000 }
gfCNCPoint5[1685] = {X 294.6527, Y 42.4586, Z -6.3333, A 0.000, B 0.000, C 0.000 }
gfCNCPoint5[1686] = {X 294.9541, Y 43.3110, Z -6.3333, A 0.000, B 0.000, C 0.000 }
gfCNCPoint5[1687] = {X 295.0611, Y 44.2089, Z -6.3333, A 0.000, B 0.000, C 0.000 }
gfCNCPoint5[1688] = {X 295.0611, Y 45.0000, Z -6.3333, A 0.000, B 0.000, C 0.000 }
gfCNCPoint5[1689] = {X 294.9608, Y 45.8901, Z -6.3333, A 0.000, B 0.000, C 0.000 }
gfCNCPoint5[1690] = {X 294.6650, Y 46.7355, Z -6.3333, A 0.000, B 0.000, C 0.000 }
gfCNCPoint5[1691] = {X 294.1885, Y 47.4940, Z -6.3333, A 0.000, B 0.000, C 0.000 }
gfCNCPoint5[1692] = {X 293.5551, Y 48.1273, Z -6.3333, A 0.000, B 0.000, C 0.000 }
gfCNCPoint5[1693] = {X 292.7967, Y 48.6039, Z -6.3333, A 0.000, B 0.000, C 0.000 }
gfCNCPoint5[1694] = {X 291.9512, Y 48.8997, Z -6.3333, A 0.000, B 0.000, C 0.000 }
gfCNCPoint5[1695] = {X 291.0611, Y 49.0000, Z -6.3333, A 0.000, B 0.000, C 0.000 }
gfCNCPoint5[1696] = {X 284.6177, Y 49.0000, Z -6.3333, A 0.000, B 0.000, C 0.000 }
gfCNCPoint5[1697] = {X 283.7276, Y 48.8997, Z -6.3333, A 0.000, B 0.000, C 0.000 }
gfCNCPoint5[1698] = {X 282.8821, Y 48.6039, Z -6.3333, A 0.000, B 0.000, C 0.000 }
gfCNCPoint5[1699] = {X 282.1237, Y 48.1273, Z -6.3333, A 0.000, B 0.000, C 0.000 }
gfCNCPoint5[1700] = {X 281.4903, Y 47.4939, Z -6.3333, A 0.000, B 0.000, C 0.000 }
gfCNCPoint5[1701] = {X 281.0138, Y 46.7355, Z -6.3333, A 0.000, B 0.000, C 0.000 }
gfCNCPoint5[1702] = {X 280.7180, Y 45.8901, Z -6.3333, A 0.000, B 0.000, C 0.000 }
gfCNCPoint5[1703] = {X 280.6177, Y 45.0000, Z -6.3333, A 0.000, B 0.000, C 0.000 }
gfCNCPoint5[1704] = {X 280.6177, Y 44.2089, Z -6.3333, A 0.000, B 0.000, C 0.000 }
gfCNCPoint5[1705] = {X 280.7225, Y 43.3124, Z -6.3333, A 0.000, B 0.000, C 0.000 }
gfCNCPoint5[1706] = {X 281.0234, Y 42.4615, Z -6.3333, A 0.000, B 0.000, C 0.000 }
gfCNCPoint5[1707] = {X 281.5055, Y 41.6985, Z -6.3333, A 0.000, B 0.000, C 0.000 }
gfCNCPoint5[1708] = {X 282.1447, Y 41.0613, Z -6.3333, A 0.000, B 0.000, C 0.000 }
gfCNCPoint5[1709] = {X 282.1445, Y 28.5920, Z -6.3333, A 0.000, B 0.000, C 0.000 }
gfCNCPoint5[1710] = {X 278.0645, Y 28.5921, Z -6.3333, A 0.000, B 0.000, C 0.000 }
gfCNCPoint5[1711] = {X 278.0645, Y 28.5921, Z -3.3333, A 0.000, B 0.000, C 0.000 }
gfCNCPoint5[1712] = {X 278.0645, Y 28.5921, Z 11.0000, A 0.000, B 0.000, C 0.000 }
gfCNCPoint5[1713] = {X 353.3539, Y 107.0412, Z 11.0000, A 0.000, B 0.000, C 0.000 }
gfCNCPoint5[1714] = {X 353.3539, Y 107.0412, Z -3.3333, A 0.000, B 0.000, C 0.000 }
gfCNCPoint5[1715] = {X 353.3539, Y 107.0412, Z -6.3333, A 0.000, B 0.000, C 0.000 }
gfCNCPoint5[1716] = {X 353.2425, Y 102.9627, Z -6.3333, A 0.000, B 0.000, C 0.000 }
gfCNCPoint5[1717] = {X 348.1837, Y 103.0326, Z -6.3333, A 0.000, B 0.000, C 0.000 }
gfCNCPoint5[1718] = {X 343.1250, Y 102.9658, Z -6.3333, A 0.000, B 0.000, C 0.000 }
gfCNCPoint5[1719] = {X 338.0698, Y 102.7625, Z -6.3333, A 0.000, B 0.000, C 0.000 }
gfCNCPoint5[1720] = {X 334.1156, Y 102.4855, Z -6.3333, A 0.000, B 0.000, C 0.000 }
gfCNCPoint5[1721] = {X 330.1763, Y 102.0437, Z -6.3333, A 0.000, B 0.000, C 0.000 }
gfCNCPoint5[1722] = {X 326.2590, Y 101.4377, Z -6.3333, A 0.000, B 0.000, C 0.000 }
gfCNCPoint5[1723] = {X 323.4095, Y 100.8331, Z -6.3333, A 0.000, B 0.000, C 0.000 }
gfCNCPoint5[1724] = {X 320.6122, Y 100.0202, Z -6.3333, A 0.000, B 0.000, C 0.000 }
gfCNCPoint5[1725] = {X 317.8824, Y 99.0034, Z -6.3333, A 0.000, B 0.000, C 0.000 }
gfCNCPoint5[1726] = {X 316.3695, Y 98.3056, Z -6.3333, A 0.000, B 0.000, C 0.000 }
gfCNCPoint5[1727] = {X 314.9202, Y 97.4837, Z -6.3333, A 0.000, B 0.000, C 0.000 }
gfCNCPoint5[1728] = {X 313.5447, Y 96.5436, Z -6.3333, A 0.000, B 0.000, C 0.000 }
gfCNCPoint5[1729] = {X 312.2527, Y 95.4917, Z -6.3333, A 0.000, B 0.000, C 0.000 }
gfCNCPoint5[1730] = {X 311.2489, Y 94.4931, Z -6.3333, A 0.000, B 0.000, C 0.000 }
gfCNCPoint5[1731] = {X 310.3706, Y 93.3825, Z -6.3333, A 0.000, B 0.000, C 0.000 }
gfCNCPoint5[1732] = {X 309.6300, Y 92.1757, Z -6.3333, A 0.000, B 0.000, C 0.000 }
gfCNCPoint5[1733] = {X 309.0377, Y 90.8896, Z -6.3333, A 0.000, B 0.000, C 0.000 }
gfCNCPoint5[1734] = {X 308.6020, Y 89.5424, Z -6.3333, A 0.000, B 0.000, C 0.000 }
gfCNCPoint5[1735] = {X 308.2585, Y 87.9192, Z -6.3333, A 0.000, B 0.000, C 0.000 }
gfCNCPoint5[1736] = {X 308.0556, Y 86.2726, Z -6.3333, A 0.000, B 0.000, C 0.000 }
gfCNCPoint5[1737] = {X 307.9947, Y 84.6147, Z -6.3333, A 0.000, B 0.000, C 0.000 }
gfCNCPoint5[1738] = {X 307.9960, Y 63.2122, Z -6.3333, A 0.000, B 0.000, C 0.000 }
gfCNCPoint5[1739] = {X 307.1445, Y 63.0029, Z -6.3333, A 0.000, B 0.000, C 0.000 }
gfCNCPoint5[1740] = {X 306.3529, Y 62.6259, Z -6.3333, A 0.000, B 0.000, C 0.000 }
gfCNCPoint5[1741] = {X 305.6537, Y 62.0970, Z -6.3333, A 0.000, B 0.000, C 0.000 }
gfCNCPoint5[1742] = {X 305.0757, Y 61.4377, Z -6.3333, A 0.000, B 0.000, C 0.000 }
gfCNCPoint5[1743] = {X 304.6427, Y 60.6753, Z -6.3333, A 0.000, B 0.000, C 0.000 }
gfCNCPoint5[1744] = {X 304.3725, Y 59.8412, Z -6.3333, A 0.000, B 0.000, C 0.000 }
gfCNCPoint5[1745] = {X 304.2764, Y 58.9697, Z -6.3333, A 0.000, B 0.000, C 0.000 }
gfCNCPoint5[1746] = {X 304.2762, Y 58.0000, Z -6.3333, A 0.000, B 0.000, C 0.000 }
gfCNCPoint5[1747] = {X 304.3845, Y 57.0387, Z -6.3333, A 0.000, B 0.000, C 0.000 }
gfCNCPoint5[1748] = {X 304.7040, Y 56.1256, Z -6.3333, A 0.000, B 0.000, C 0.000 }
gfCNCPoint5[1749] = {X 305.2187, Y 55.3065, Z -6.3333, A 0.000, B 0.000, C 0.000 }
gfCNCPoint5[1750] = {X 305.9027, Y 54.6225, Z -6.3333, A 0.000, B 0.000, C 0.000 }
gfCNCPoint5[1751] = {X 306.7218, Y 54.1078, Z -6.3333, A 0.000, B 0.000, C 0.000 }
gfCNCPoint5[1752] = {X 307.6349, Y 53.7883, Z -6.3333, A 0.000, B 0.000, C 0.000 }
gfCNCPoint5[1753] = {X 308.5962, Y 53.6800, Z -6.3333, A 0.000, B 0.000, C 0.000 }
gfCNCPoint5[1754] = {X 324.3107, Y 53.6800, Z -6.3333, A 0.000, B 0.000, C 0.000 }
gfCNCPoint5[1755] = {X 325.2720, Y 53.7883, Z -6.3333, A 0.000, B 0.000, C 0.000 }
gfCNCPoint5[1756] = {X 326.1851, Y 54.1078, Z -6.3333, A 0.000, B 0.000, C 0.000 }
gfCNCPoint5[1757] = {X 327.0042, Y 54.6225, Z -6.3333, A 0.000, B 0.000, C 0.000 }
gfCNCPoint5[1758] = {X 327.6882, Y 55.3065, Z -6.3333, A 0.000, B 0.000, C 0.000 }
gfCNCPoint5[1759] = {X 328.2029, Y 56.1256, Z -6.3333, A 0.000, B 0.000, C 0.000 }
gfCNCPoint5[1760] = {X 328.5224, Y 57.0387, Z -6.3333, A 0.000, B 0.000, C 0.000 }
gfCNCPoint5[1761] = {X 328.6307, Y 58.0000, Z -6.3333, A 0.000, B 0.000, C 0.000 }
gfCNCPoint5[1762] = {X 328.6307, Y 58.9358, Z -6.3333, A 0.000, B 0.000, C 0.000 }
gfCNCPoint5[1763] = {X 328.5368, Y 59.8122, Z -6.3333, A 0.000, B 0.000, C 0.000 }
gfCNCPoint5[1764] = {X 328.2685, Y 60.6517, Z -6.3333, A 0.000, B 0.000, C 0.000 }
gfCNCPoint5[1765] = {X 327.8368, Y 61.4201, Z -6.3333, A 0.000, B 0.000, C 0.000 }
gfCNCPoint5[1766] = {X 327.2592, Y 62.0859, Z -6.3333, A 0.000, B 0.000, C 0.000 }
gfCNCPoint5[1767] = {X 326.5596, Y 62.6218, Z -6.3333, A 0.000, B 0.000, C 0.000 }
gfCNCPoint5[1768] = {X 325.7664, Y 63.0060, Z -6.3333, A 0.000, B 0.000, C 0.000 }
gfCNCPoint5[1769] = {X 324.9121, Y 63.2228, Z -6.3333, A 0.000, B 0.000, C 0.000 }
gfCNCPoint5[1770] = {X 324.9139, Y 83.2295, Z -6.3333, A 0.000, B 0.000, C 0.000 }
gfCNCPoint5[1771] = {X 324.9274, Y 84.6146, Z -6.3333, A 0.000, B 0.000, C 0.000 }
gfCNCPoint5[1772] = {X 325.0049, Y 85.8497, Z -6.3333, A 0.000, B 0.000, C 0.000 }
gfCNCPoint5[1773] = {X 325.2262, Y 87.0672, Z -6.3333, A 0.000, B 0.000, C 0.000 }
gfCNCPoint5[1774] = {X 325.4716, Y 87.3357, Z -6.3333, A 0.000, B 0.000, C 0.000 }
gfCNCPoint5[1775] = {X 325.7737, Y 87.5382, Z -6.3333, A 0.000, B 0.000, C 0.000 }
gfCNCPoint5[1776] = {X 326.2253, Y 87.7937, Z -6.3333, A 0.000, B 0.000, C 0.000 }
gfCNCPoint5[1777] = {X 327.6628, Y 88.3900, Z -6.3333, A 0.000, B 0.000, C 0.000 }
gfCNCPoint5[1778] = {X 329.1569, Y 88.8253, Z -6.3333, A 0.000, B 0.000, C 0.000 }
gfCNCPoint5[1779] = {X 331.4311, Y 89.2988, Z -6.3333, A 0.000, B 0.000, C 0.000 }
gfCNCPoint5[1780] = {X 333.7258, Y 89.6600, Z -6.3333, A 0.000, B 0.000, C 0.000 }
gfCNCPoint5[1781] = {X 336.0355, Y 89.9080, Z -6.3333, A 0.000, B 0.000, C 0.000 }
gfCNCPoint5[1782] = {X 340.4056, Y 90.2022, Z -6.3333, A 0.000, B 0.000, C 0.000 }
gfCNCPoint5[1783] = {X 344.7828, Y 90.3561, Z -6.3333, A 0.000, B 0.000, C 0.000 }
gfCNCPoint5[1784] = {X 349.1628, Y 90.3693, Z -6.3333, A 0.000, B 0.000, C 0.000 }
gfCNCPoint5[1785] = {X 353.3143, Y 90.3010, Z -6.3333, A 0.000, B 0.000, C 0.000 }
gfCNCPoint5[1786] = {X 357.4606, Y 90.0821, Z -6.3333, A 0.000, B 0.000, C 0.000 }
gfCNCPoint5[1787] = {X 361.5962, Y 89.7127, Z -6.3333, A 0.000, B 0.000, C 0.000 }
gfCNCPoint5[1788] = {X 363.6775, Y 89.4256, Z -6.3333, A 0.000, B 0.000, C 0.000 }
gfCNCPoint5[1789] = {X 365.7396, Y 89.0236, Z -6.3333, A 0.000, B 0.000, C 0.000 }
gfCNCPoint5[1790] = {X 367.7763, Y 88.5079, Z -6.3333, A 0.000, B 0.000, C 0.000 }
gfCNCPoint5[1791] = {X 368.7082, Y 88.1948, Z -6.3333, A 0.000, B 0.000, C 0.000 }
gfCNCPoint5[1792] = {X 369.5991, Y 87.7790, Z -6.3333, A 0.000, B 0.000, C 0.000 }
gfCNCPoint5[1793] = {X 370.4378, Y 87.2660, Z -6.3333, A 0.000, B 0.000, C 0.000 }
gfCNCPoint5[1794] = {X 370.5874, Y 87.1103, Z -6.3333, A 0.000, B 0.000, C 0.000 }
gfCNCPoint5[1795] = {X 370.6646, Y 86.9086, Z -6.3333, A 0.000, B 0.000, C 0.000 }
gfCNCPoint5[1796] = {X 370.8556, Y 85.3739, Z -6.3333, A 0.000, B 0.000, C 0.000 }
gfCNCPoint5[1797] = {X 370.9194, Y 83.8287, Z -6.3333, A 0.000, B 0.000, C 0.000 }
gfCNCPoint5[1798] = {X 370.9201, Y 63.2123, Z -6.3333, A 0.000, B 0.000, C 0.000 }
gfCNCPoint5[1799] = {X 370.0685, Y 63.0032, Z -6.3333, A 0.000, B 0.000, C 0.000 }
gfCNCPoint5[1800] = {X 369.2767, Y 62.6264, Z -6.3333, A 0.000, B 0.000, C 0.000 }
gfCNCPoint5[1801] = {X 368.5772, Y 62.0974, Z -6.3333, A 0.000, B 0.000, C 0.000 }
gfCNCPoint5[1802] = {X 367.9990, Y 61.4381, Z -6.3333, A 0.000, B 0.000, C 0.000 }
gfCNCPoint5[1803] = {X 367.5659, Y 60.6756, Z -6.3333, A 0.000, B 0.000, C 0.000 }
gfCNCPoint5[1804] = {X 367.2956, Y 59.8414, Z -6.3333, A 0.000, B 0.000, C 0.000 }
gfCNCPoint5[1805] = {X 367.1994, Y 58.9697, Z -6.3333, A 0.000, B 0.000, C 0.000 }
gfCNCPoint5[1806] = {X 367.1993, Y 58.0000, Z -6.3333, A 0.000, B 0.000, C 0.000 }
gfCNCPoint5[1807] = {X 367.3076, Y 57.0387, Z -6.3333, A 0.000, B 0.000, C 0.000 }
gfCNCPoint5[1808] = {X 367.6271, Y 56.1256, Z -6.3333, A 0.000, B 0.000, C 0.000 }
gfCNCPoint5[1809] = {X 368.1418, Y 55.3065, Z -6.3333, A 0.000, B 0.000, C 0.000 }
gfCNCPoint5[1810] = {X 368.8258, Y 54.6225, Z -6.3333, A 0.000, B 0.000, C 0.000 }
gfCNCPoint5[1811] = {X 369.6449, Y 54.1078, Z -6.3333, A 0.000, B 0.000, C 0.000 }
gfCNCPoint5[1812] = {X 370.5580, Y 53.7883, Z -6.3333, A 0.000, B 0.000, C 0.000 }
gfCNCPoint5[1813] = {X 371.5193, Y 53.6800, Z -6.3333, A 0.000, B 0.000, C 0.000 }
gfCNCPoint5[1814] = {X 388.0597, Y 53.6800, Z -6.3333, A 0.000, B 0.000, C 0.000 }
gfCNCPoint5[1815] = {X 389.0210, Y 53.7883, Z -6.3333, A 0.000, B 0.000, C 0.000 }
gfCNCPoint5[1816] = {X 389.9341, Y 54.1078, Z -6.3333, A 0.000, B 0.000, C 0.000 }
gfCNCPoint5[1817] = {X 390.7532, Y 54.6225, Z -6.3333, A 0.000, B 0.000, C 0.000 }
gfCNCPoint5[1818] = {X 391.4372, Y 55.3065, Z -6.3333, A 0.000, B 0.000, C 0.000 }
gfCNCPoint5[1819] = {X 391.9519, Y 56.1256, Z -6.3333, A 0.000, B 0.000, C 0.000 }
gfCNCPoint5[1820] = {X 392.2714, Y 57.0387, Z -6.3333, A 0.000, B 0.000, C 0.000 }
gfCNCPoint5[1821] = {X 392.3797, Y 58.0000, Z -6.3333, A 0.000, B 0.000, C 0.000 }
gfCNCPoint5[1822] = {X 392.3797, Y 58.9342, Z -6.3333, A 0.000, B 0.000, C 0.000 }
gfCNCPoint5[1823] = {X 392.2673, Y 59.9128, Z -6.3333, A 0.000, B 0.000, C 0.000 }
gfCNCPoint5[1824] = {X 391.9363, Y 60.8405, Z -6.3333, A 0.000, B 0.000, C 0.000 }
gfCNCPoint5[1825] = {X 391.4939, Y 61.5569, Z -6.3333, A 0.000, B 0.000, C 0.000 }
gfCNCPoint5[1826] = {X 390.9216, Y 62.1745, Z -6.3333, A 0.000, B 0.000, C 0.000 }
gfCNCPoint5[1827] = {X 390.2408, Y 62.6700, Z -6.3333, A 0.000, B 0.000, C 0.000 }
gfCNCPoint5[1828] = {X 389.4773, Y 63.0249, Z -6.3333, A 0.000, B 0.000, C 0.000 }
gfCNCPoint5[1829] = {X 388.6596, Y 63.2258, Z -6.3333, A 0.000, B 0.000, C 0.000 }
gfCNCPoint5[1830] = {X 388.6576, Y 84.6147, Z -6.3333, A 0.000, B 0.000, C 0.000 }
gfCNCPoint5[1831] = {X 388.5977, Y 86.2731, Z -6.3333, A 0.000, B 0.000, C 0.000 }
gfCNCPoint5[1832] = {X 388.3934, Y 87.9199, Z -6.3333, A 0.000, B 0.000, C 0.000 }
gfCNCPoint5[1833] = {X 388.0461, Y 89.5425, Z -6.3333, A 0.000, B 0.000, C 0.000 }
gfCNCPoint5[1834] = {X 387.5139, Y 91.1298, Z -6.3333, A 0.000, B 0.000, C 0.000 }
gfCNCPoint5[1835] = {X 386.7643, Y 92.6268, Z -6.3333, A 0.000, B 0.000, C 0.000 }
gfCNCPoint5[1836] = {X 385.8123, Y 94.0038, Z -6.3333, A 0.000, B 0.000, C 0.000 }
gfCNCPoint5[1837] = {X 384.6765, Y 95.2337, Z -6.3333, A 0.000, B 0.000, C 0.000 }
gfCNCPoint5[1838] = {X 383.1619, Y 96.5102, Z -6.3333, A 0.000, B 0.000, C 0.000 }
gfCNCPoint5[1839] = {X 381.5203, Y 97.6185, Z -6.3333, A 0.000, B 0.000, C 0.000 }
gfCNCPoint5[1840] = {X 379.7703, Y 98.5463, Z -6.3333, A 0.000, B 0.000, C 0.000 }
gfCNCPoint5[1841] = {X 377.4988, Y 99.5012, Z -6.3333, A 0.000, B 0.000, C 0.000 }
gfCNCPoint5[1842] = {X 375.1648, Y 100.2915, Z -6.3333, A 0.000, B 0.000, C 0.000 }
gfCNCPoint5[1843] = {X 372.7804, Y 100.9129, Z -6.3333, A 0.000, B 0.000, C 0.000 }
gfCNCPoint5[1844] = {X 368.8697, Y 101.6670, Z -6.3333, A 0.000, B 0.000, C 0.000 }
gfCNCPoint5[1845] = {X 364.9265, Y 102.2273, Z -6.3333, A 0.000, B 0.000, C 0.000 }
gfCNCPoint5[1846] = {X 360.9605, Y 102.5925, Z -6.3333, A 0.000, B 0.000, C 0.000 }
gfCNCPoint5[1847] = {X 357.1034, Y 102.8174, Z -6.3333, A 0.000, B 0.000, C 0.000 }
gfCNCPoint5[1848] = {X 353.2425, Y 102.9627, Z -6.3333, A 0.000, B 0.000, C 0.000 }
gfCNCPoint5[1849] = {X 353.3517, Y 106.9612, Z -6.3333, A 0.000, B 0.000, C 0.000 }
gfCNCPoint5[1850] = {X 353.2403, Y 102.8828, Z -6.3333, A 0.000, B 0.000, C 0.000 }
gfCNCPoint5[1851] = {X 348.1837, Y 102.9526, Z -6.3333, A 0.000, B 0.000, C 0.000 }
gfCNCPoint5[1852] = {X 343.1270, Y 102.8859, Z -6.3333, A 0.000, B 0.000, C 0.000 }
gfCNCPoint5[1853] = {X 338.0740, Y 102.6826, Z -6.3333, A 0.000, B 0.000, C 0.000 }
gfCNCPoint5[1854] = {X 334.1230, Y 102.4059, Z -6.3333, A 0.000, B 0.000, C 0.000 }
gfCNCPoint5[1855] = {X 330.1870, Y 101.9644, Z -6.3333, A 0.000, B 0.000, C 0.000 }
gfCNCPoint5[1856] = {X 326.2729, Y 101.3589, Z -6.3333, A 0.000, B 0.000, C 0.000 }
gfCNCPoint5[1857] = {X 323.4290, Y 100.7555, Z -6.3333, A 0.000, B 0.000, C 0.000 }
gfCNCPoint5[1858] = {X 320.6373, Y 99.9442, Z -6.3333, A 0.000, B 0.000, C 0.000 }
gfCNCPoint5[1859] = {X 317.9130, Y 98.9294, Z -6.3333, A 0.000, B 0.000, C 0.000 }
gfCNCPoint5[1860] = {X 316.4061, Y 98.2344, Z -6.3333, A 0.000, B 0.000, C 0.000 }
gfCNCPoint5[1861] = {X 314.9626, Y 97.4159, Z -6.3333, A 0.000, B 0.000, C 0.000 }
gfCNCPoint5[1862] = {X 313.5926, Y 96.4795, Z -6.3333, A 0.000, B 0.000, C 0.000 }
gfCNCPoint5[1863] = {X 312.3057, Y 95.4318, Z -6.3333, A 0.000, B 0.000, C 0.000 }
gfCNCPoint5[1864] = {X 311.3086, Y 94.4398, Z -6.3333, A 0.000, B 0.000, C 0.000 }
gfCNCPoint5[1865] = {X 310.4362, Y 93.3367, Z -6.3333, A 0.000, B 0.000, C 0.000 }
gfCNCPoint5[1866] = {X 309.7006, Y 92.1380, Z -6.3333, A 0.000, B 0.000, C 0.000 }
gfCNCPoint5[1867] = {X 309.1122, Y 90.8605, Z -6.3333, A 0.000, B 0.000, C 0.000 }
gfCNCPoint5[1868] = {X 308.6794, Y 89.5223, Z -6.3333, A 0.000, B 0.000, C 0.000 }
gfCNCPoint5[1869] = {X 308.3374, Y 87.9059, Z -6.3333, A 0.000, B 0.000, C 0.000 }
gfCNCPoint5[1870] = {X 308.1353, Y 86.2661, Z -6.3333, A 0.000, B 0.000, C 0.000 }
gfCNCPoint5[1871] = {X 308.0747, Y 84.6150, Z -6.3333, A 0.000, B 0.000, C 0.000 }
gfCNCPoint5[1872] = {X 308.0760, Y 63.1420, Z -6.3333, A 0.000, B 0.000, C 0.000 }
gfCNCPoint5[1873] = {X 307.2277, Y 62.9471, Z -6.3333, A 0.000, B 0.000, C 0.000 }
gfCNCPoint5[1874] = {X 306.4370, Y 62.5831, Z -6.3333, A 0.000, B 0.000, C 0.000 }
gfCNCPoint5[1875] = {X 305.7374, Y 62.0653, Z -6.3333, A 0.000, B 0.000, C 0.000 }
gfCNCPoint5[1876] = {X 305.1582, Y 61.4156, Z -6.3333, A 0.000, B 0.000, C 0.000 }
gfCNCPoint5[1877] = {X 304.7240, Y 60.6612, Z -6.3333, A 0.000, B 0.000, C 0.000 }
gfCNCPoint5[1878] = {X 304.4529, Y 59.8341, Z -6.3333, A 0.000, B 0.000, C 0.000 }
gfCNCPoint5[1879] = {X 304.3564, Y 58.9691, Z -6.3333, A 0.000, B 0.000, C 0.000 }
gfCNCPoint5[1880] = {X 304.3562, Y 58.0000, Z -6.3333, A 0.000, B 0.000, C 0.000 }
gfCNCPoint5[1881] = {X 304.4625, Y 57.0565, Z -6.3333, A 0.000, B 0.000, C 0.000 }
gfCNCPoint5[1882] = {X 304.7761, Y 56.1603, Z -6.3333, A 0.000, B 0.000, C 0.000 }
gfCNCPoint5[1883] = {X 305.2813, Y 55.3564, Z -6.3333, A 0.000, B 0.000, C 0.000 }
gfCNCPoint5[1884] = {X 305.9526, Y 54.6850, Z -6.3333, A 0.000, B 0.000, C 0.000 }
gfCNCPoint5[1885] = {X 306.7566, Y 54.1799, Z -6.3333, A 0.000, B 0.000, C 0.000 }
gfCNCPoint5[1886] = {X 307.6527, Y 53.8663, Z -6.3333, A 0.000, B 0.000, C 0.000 }
gfCNCPoint5[1887] = {X 308.5962, Y 53.7600, Z -6.3333, A 0.000, B 0.000, C 0.000 }
gfCNCPoint5[1888] = {X 324.3107, Y 53.7600, Z -6.3333, A 0.000, B 0.000, C 0.000 }
gfCNCPoint5[1889] = {X 325.2542, Y 53.8663, Z -6.3333, A 0.000, B 0.000, C 0.000 }
gfCNCPoint5[1890] = {X 326.1504, Y 54.1799, Z -6.3333, A 0.000, B 0.000, C 0.000 }
gfCNCPoint5[1891] = {X 326.9543, Y 54.6850, Z -6.3333, A 0.000, B 0.000, C 0.000 }
gfCNCPoint5[1892] = {X 327.6257, Y 55.3564, Z -6.3333, A 0.000, B 0.000, C 0.000 }
gfCNCPoint5[1893] = {X 328.1308, Y 56.1603, Z -6.3333, A 0.000, B 0.000, C 0.000 }
gfCNCPoint5[1894] = {X 328.4444, Y 57.0565, Z -6.3333, A 0.000, B 0.000, C 0.000 }
gfCNCPoint5[1895] = {X 328.5507, Y 58.0000, Z -6.3333, A 0.000, B 0.000, C 0.000 }
gfCNCPoint5[1896] = {X 328.5507, Y 58.9354, Z -6.3333, A 0.000, B 0.000, C 0.000 }
gfCNCPoint5[1897] = {X 328.4565, Y 59.8053, Z -6.3333, A 0.000, B 0.000, C 0.000 }
gfCNCPoint5[1898] = {X 328.1873, Y 60.6378, Z -6.3333, A 0.000, B 0.000, C 0.000 }
gfCNCPoint5[1899] = {X 327.7543, Y 61.3981, Z -6.3333, A 0.000, B 0.000, C 0.000 }
gfCNCPoint5[1900] = {X 327.1756, Y 62.0545, Z -6.3333, A 0.000, B 0.000, C 0.000 }
gfCNCPoint5[1901] = {X 326.4755, Y 62.5793, Z -6.3333, A 0.000, B 0.000, C 0.000 }
gfCNCPoint5[1902] = {X 325.6833, Y 62.9507, Z -6.3333, A 0.000, B 0.000, C 0.000 }
gfCNCPoint5[1903] = {X 324.8321, Y 63.1532, Z -6.3333, A 0.000, B 0.000, C 0.000 }
gfCNCPoint5[1904] = {X 324.8339, Y 83.2300, Z -6.3333, A 0.000, B 0.000, C 0.000 }
gfCNCPoint5[1905] = {X 324.8474, Y 84.6149, Z -6.3333, A 0.000, B 0.000, C 0.000 }
gfCNCPoint5[1906] = {X 324.9264, Y 85.8670, Z -6.3333, A 0.000, B 0.000, C 0.000 }
gfCNCPoint5[1907] = {X 325.1521, Y 87.1010, Z -6.3333, A 0.000, B 0.000, C 0.000 }
gfCNCPoint5[1908] = {X 325.4128, Y 87.3906, Z -6.3333, A 0.000, B 0.000, C 0.000 }
gfCNCPoint5[1909] = {X 325.7358, Y 87.6087, Z -6.3333, A 0.000, B 0.000, C 0.000 }
gfCNCPoint5[1910] = {X 326.1882, Y 87.8647, Z -6.3333, A 0.000, B 0.000, C 0.000 }
gfCNCPoint5[1911] = {X 327.6349, Y 88.4650, Z -6.3333, A 0.000, B 0.000, C 0.000 }
gfCNCPoint5[1912] = {X 329.1387, Y 88.9033, Z -6.3333, A 0.000, B 0.000, C 0.000 }
gfCNCPoint5[1913] = {X 331.4168, Y 89.3775, Z -6.3333, A 0.000, B 0.000, C 0.000 }
gfCNCPoint5[1914] = {X 333.7153, Y 89.7393, Z -6.3333, A 0.000, B 0.000, C 0.000 }
gfCNCPoint5[1915] = {X 336.0289, Y 89.9877, Z -6.3333, A 0.000, B 0.000, C 0.000 }
gfCNCPoint5[1916] = {X 340.4015, Y 90.2821, Z -6.3333, A 0.000, B 0.000, C 0.000 }
gfCNCPoint5[1917] = {X 344.7813, Y 90.4361, Z -6.3333, A 0.000, B 0.000, C 0.000 }
gfCNCPoint5[1918] = {X 349.1638, Y 90.4493, Z -6.3333, A 0.000, B 0.000, C 0.000 }
gfCNCPoint5[1919] = {X 353.3179, Y 90.3809, Z -6.3333, A 0.000, B 0.000, C 0.000 }
gfCNCPoint5[1920] = {X 357.4667, Y 90.1618, Z -6.3333, A 0.000, B 0.000, C 0.000 }
gfCNCPoint5[1921] = {X 361.6049, Y 89.7922, Z -6.3333, A 0.000, B 0.000, C 0.000 }
gfCNCPoint5[1922] = {X 363.6906, Y 89.5045, Z -6.3333, A 0.000, B 0.000, C 0.000 }
gfCNCPoint5[1923] = {X 365.7571, Y 89.1017, Z -6.3333, A 0.000, B 0.000, C 0.000 }
gfCNCPoint5[1924] = {X 367.7981, Y 88.5849, Z -6.3333, A 0.000, B 0.000, C 0.000 }
gfCNCPoint5[1925] = {X 368.7383, Y 88.2689, Z -6.3333, A 0.000, B 0.000, C 0.000 }
gfCNCPoint5[1926] = {X 369.6372, Y 87.8494, Z -6.3333, A 0.000, B 0.000, C 0.000 }
gfCNCPoint5[1927] = {X 370.4833, Y 87.3318, Z -6.3333, A 0.000, B 0.000, C 0.000 }
gfCNCPoint5[1928] = {X 370.6550, Y 87.1532, Z -6.3333, A 0.000, B 0.000, C 0.000 }
gfCNCPoint5[1929] = {X 370.7435, Y 86.9218, Z -6.3333, A 0.000, B 0.000, C 0.000 }
gfCNCPoint5[1930] = {X 370.9354, Y 85.3805, Z -6.3333, A 0.000, B 0.000, C 0.000 }
gfCNCPoint5[1931] = {X 370.9994, Y 83.8287, Z -6.3333, A 0.000, B 0.000, C 0.000 }
gfCNCPoint5[1932] = {X 371.0001, Y 63.1422, Z -6.3333, A 0.000, B 0.000, C 0.000 }
gfCNCPoint5[1933] = {X 370.1516, Y 62.9474, Z -6.3333, A 0.000, B 0.000, C 0.000 }
gfCNCPoint5[1934] = {X 369.3608, Y 62.5835, Z -6.3333, A 0.000, B 0.000, C 0.000 }
gfCNCPoint5[1935] = {X 368.6609, Y 62.0657, Z -6.3333, A 0.000, B 0.000, C 0.000 }
gfCNCPoint5[1936] = {X 368.0816, Y 61.4159, Z -6.3333, A 0.000, B 0.000, C 0.000 }
gfCNCPoint5[1937] = {X 367.6471, Y 60.6615, Z -6.3333, A 0.000, B 0.000, C 0.000 }
gfCNCPoint5[1938] = {X 367.3759, Y 59.8343, Z -6.3333, A 0.000, B 0.000, C 0.000 }
gfCNCPoint5[1939] = {X 367.2794, Y 58.9691, Z -6.3333, A 0.000, B 0.000, C 0.000 }
gfCNCPoint5[1940] = {X 367.2793, Y 58.0000, Z -6.3333, A 0.000, B 0.000, C 0.000 }
gfCNCPoint5[1941] = {X 367.3856, Y 57.0565, Z -6.3333, A 0.000, B 0.000, C 0.000 }
gfCNCPoint5[1942] = {X 367.6992, Y 56.1603, Z -6.3333, A 0.000, B 0.000, C 0.000 }
gfCNCPoint5[1943] = {X 368.2043, Y 55.3564, Z -6.3333, A 0.000, B 0.000, C 0.000 }
gfCNCPoint5[1944] = {X 368.8757, Y 54.6850, Z -6.3333, A 0.000, B 0.000, C 0.000 }
gfCNCPoint5[1945] = {X 369.6796, Y 54.1799, Z -6.3333, A 0.000, B 0.000, C 0.000 }
gfCNCPoint5[1946] = {X 370.5758, Y 53.8663, Z -6.3333, A 0.000, B 0.000, C 0.000 }
gfCNCPoint5[1947] = {X 371.5193, Y 53.7600, Z -6.3333, A 0.000, B 0.000, C 0.000 }
gfCNCPoint5[1948] = {X 388.0597, Y 53.7600, Z -6.3333, A 0.000, B 0.000, C 0.000 }
gfCNCPoint5[1949] = {X 389.0032, Y 53.8663, Z -6.3333, A 0.000, B 0.000, C 0.000 }
gfCNCPoint5[1950] = {X 389.8993, Y 54.1799, Z -6.3333, A 0.000, B 0.000, C 0.000 }
gfCNCPoint5[1951] = {X 390.7033, Y 54.6850, Z -6.3333, A 0.000, B 0.000, C 0.000 }
gfCNCPoint5[1952] = {X 391.3746, Y 55.3564, Z -6.3333, A 0.000, B 0.000, C 0.000 }
gfCNCPoint5[1953] = {X 391.8798, Y 56.1603, Z -6.3333, A 0.000, B 0.000, C 0.000 }
gfCNCPoint5[1954] = {X 392.1934, Y 57.0565, Z -6.3333, A 0.000, B 0.000, C 0.000 }
gfCNCPoint5[1955] = {X 392.2997, Y 58.0000, Z -6.3333, A 0.000, B 0.000, C 0.000 }
gfCNCPoint5[1956] = {X 392.2997, Y 58.9342, Z -6.3333, A 0.000, B 0.000, C 0.000 }
gfCNCPoint5[1957] = {X 392.1894, Y 59.8947, Z -6.3333, A 0.000, B 0.000, C 0.000 }
gfCNCPoint5[1958] = {X 391.8645, Y 60.8052, Z -6.3333, A 0.000, B 0.000, C 0.000 }
gfCNCPoint5[1959] = {X 391.4218, Y 61.5194, Z -6.3333, A 0.000, B 0.000, C 0.000 }
gfCNCPoint5[1960] = {X 390.8477, Y 62.1329, Z -6.3333, A 0.000, B 0.000, C 0.000 }
gfCNCPoint5[1961] = {X 390.1644, Y 62.6219, Z -6.3333, A 0.000, B 0.000, C 0.000 }
gfCNCPoint5[1962] = {X 389.3985, Y 62.9674, Z -6.3333, A 0.000, B 0.000, C 0.000 }
gfCNCPoint5[1963] = {X 388.5796, Y 63.1560, Z -6.3333, A 0.000, B 0.000, C 0.000 }
gfCNCPoint5[1964] = {X 388.5776, Y 84.6151, Z -6.3333, A 0.000, B 0.000, C 0.000 }
gfCNCPoint5[1965] = {X 388.5180, Y 86.2665, Z -6.3333, A 0.000, B 0.000, C 0.000 }
gfCNCPoint5[1966] = {X 388.3145, Y 87.9065, Z -6.3333, A 0.000, B 0.000, C 0.000 }
gfCNCPoint5[1967] = {X 387.9687, Y 89.5224, Z -6.3333, A 0.000, B 0.000, C 0.000 }
gfCNCPoint5[1968] = {X 387.4401, Y 91.0990, Z -6.3333, A 0.000, B 0.000, C 0.000 }
gfCNCPoint5[1969] = {X 386.6955, Y 92.5860, Z -6.3333, A 0.000, B 0.000, C 0.000 }
gfCNCPoint5[1970] = {X 385.7499, Y 93.9538, Z -6.3333, A 0.000, B 0.000, C 0.000 }
gfCNCPoint5[1971] = {X 384.6217, Y 95.1755, Z -6.3333, A 0.000, B 0.000, C 0.000 }
gfCNCPoint5[1972] = {X 383.1136, Y 96.4464, Z -6.3333, A 0.000, B 0.000, C 0.000 }
gfCNCPoint5[1973] = {X 381.4791, Y 97.5500, Z -6.3333, A 0.000, B 0.000, C 0.000 }
gfCNCPoint5[1974] = {X 379.7366, Y 98.4737, Z -6.3333, A 0.000, B 0.000, C 0.000 }
gfCNCPoint5[1975] = {X 377.4704, Y 99.4264, Z -6.3333, A 0.000, B 0.000, C 0.000 }
gfCNCPoint5[1976] = {X 375.1419, Y 100.2148, Z -6.3333, A 0.000, B 0.000, C 0.000 }
gfCNCPoint5[1977] = {X 372.7630, Y 100.8348, Z -6.3333, A 0.000, B 0.000, C 0.000 }
gfCNCPoint5[1978] = {X 368.8562, Y 101.5881, Z -6.3333, A 0.000, B 0.000, C 0.000 }
gfCNCPoint5[1979] = {X 364.9170, Y 102.1479, Z -6.3333, A 0.000, B 0.000, C 0.000 }
gfCNCPoint5[1980] = {X 360.9550, Y 102.5126, Z -6.3333, A 0.000, B 0.000, C 0.000 }
gfCNCPoint5[1981] = {X 357.0996, Y 102.7375, Z -6.3333, A 0.000, B 0.000, C 0.000 }
gfCNCPoint5[1982] = {X 353.2403, Y 102.8828, Z -6.3333, A 0.000, B 0.000, C 0.000 }
gfCNCPoint5[1983] = {X 353.3495, Y 106.8813, Z -6.3333, A 0.000, B 0.000, C 0.000 }
gfCNCPoint5[1984] = {X 353.2381, Y 102.8028, Z -6.3333, A 0.000, B 0.000, C 0.000 }
gfCNCPoint5[1985] = {X 348.1836, Y 102.8726, Z -6.3333, A 0.000, B 0.000, C 0.000 }
gfCNCPoint5[1986] = {X 343.1291, Y 102.8059, Z -6.3333, A 0.000, B 0.000, C 0.000 }
gfCNCPoint5[1987] = {X 338.0782, Y 102.6027, Z -6.3333, A 0.000, B 0.000, C 0.000 }
gfCNCPoint5[1988] = {X 334.1304, Y 102.3262, Z -6.3333, A 0.000, B 0.000, C 0.000 }
gfCNCPoint5[1989] = {X 330.1977, Y 101.8851, Z -6.3333, A 0.000, B 0.000, C 0.000 }
gfCNCPoint5[1990] = {X 326.2868, Y 101.2801, Z -6.3333, A 0.000, B 0.000, C 0.000 }
gfCNCPoint5[1991] = {X 323.4485, Y 100.6779, Z -6.3333, A 0.000, B 0.000, C 0.000 }
gfCNCPoint5[1992] = {X 320.6624, Y 99.8682, Z -6.3333, A 0.000, B 0.000, C 0.000 }
gfCNCPoint5[1993] = {X 317.9435, Y 98.8555, Z -6.3333, A 0.000, B 0.000, C 0.000 }
gfCNCPoint5[1994] = {X 316.4427, Y 98.1633, Z -6.3333, A 0.000, B 0.000, C 0.000 }
gfCNCPoint5[1995] = {X 315.0050, Y 97.3480, Z -6.3333, A 0.000, B 0.000, C 0.000 }
gfCNCPoint5[1996] = {X 313.6405, Y 96.4154, Z -6.3333, A 0.000, B 0.000, C 0.000 }
gfCNCPoint5[1997] = {X 312.3587, Y 95.3719, Z -6.3333, A 0.000, B 0.000, C 0.000 }
gfCNCPoint5[1998] = {X 311.3684, Y 94.3867, Z -6.3333, A 0.000, B 0.000, C 0.000 }
gfCNCPoint5[1999] = {X 310.5018, Y 93.2910, Z -6.3333, A 0.000, B 0.000, C 0.000 }
gfCNCPoint5[2000] = {X 309.7712, Y 92.1003, Z -6.3333, A 0.000, B 0.000, C 0.000 }
gfCNCPoint5[2001] = {X 309.1868, Y 90.8314, Z -6.3333, A 0.000, B 0.000, C 0.000 }
gfCNCPoint5[2002] = {X 308.7569, Y 89.5022, Z -6.3333, A 0.000, B 0.000, C 0.000 }
gfCNCPoint5[2003] = {X 308.4163, Y 87.8925, Z -6.3333, A 0.000, B 0.000, C 0.000 }
gfCNCPoint5[2004] = {X 308.2151, Y 86.2596, Z -6.3333, A 0.000, B 0.000, C 0.000 }
gfCNCPoint5[2005] = {X 308.1547, Y 84.6153, Z -6.3333, A 0.000, B 0.000, C 0.000 }
gfCNCPoint5[2006] = {X 308.1560, Y 63.0707, Z -6.3333, A 0.000, B 0.000, C 0.000 }
gfCNCPoint5[2007] = {X 307.3109, Y 62.8905, Z -6.3333, A 0.000, B 0.000, C 0.000 }
gfCNCPoint5[2008] = {X 306.5214, Y 62.5397, Z -6.3333, A 0.000, B 0.000, C 0.000 }
gfCNCPoint5[2009] = {X 305.8213, Y 62.0333, Z -6.3333, A 0.000, B 0.000, C 0.000 }
gfCNCPoint5[2010] = {X 305.2409, Y 61.3932, Z -6.3333, A 0.000, B 0.000, C 0.000 }
gfCNCPoint5[2011] = {X 304.8053, Y 60.6471, Z -6.3333, A 0.000, B 0.000, C 0.000 }
gfCNCPoint5[2012] = {X 304.5332, Y 59.8270, Z -6.3333, A 0.000, B 0.000, C 0.000 }
gfCNCPoint5[2013] = {X 304.4364, Y 58.9684, Z -6.3333, A 0.000, B 0.000, C 0.000 }
gfCNCPoint5[2014] = {X 304.4362, Y 58.0000, Z -6.3333, A 0.000, B 0.000, C 0.000 }
gfCNCPoint5[2015] = {X 304.5405, Y 57.0743, Z -6.3333, A 0.000, B 0.000, C 0.000 }
gfCNCPoint5[2016] = {X 304.8482, Y 56.1950, Z -6.3333, A 0.000, B 0.000, C 0.000 }
gfCNCPoint5[2017] = {X 305.3438, Y 55.4063, Z -6.3333, A 0.000, B 0.000, C 0.000 }
gfCNCPoint5[2018] = {X 306.0025, Y 54.7476, Z -6.3333, A 0.000, B 0.000, C 0.000 }
gfCNCPoint5[2019] = {X 306.7913, Y 54.2520, Z -6.3333, A 0.000, B 0.000, C 0.000 }
gfCNCPoint5[2020] = {X 307.6705, Y 53.9443, Z -6.3333, A 0.000, B 0.000, C 0.000 }
gfCNCPoint5[2021] = {X 308.5962, Y 53.8400, Z -6.3333, A 0.000, B 0.000, C 0.000 }
gfCNCPoint5[2022] = {X 324.3107, Y 53.8400, Z -6.3333, A 0.000, B 0.000, C 0.000 }
gfCNCPoint5[2023] = {X 325.2364, Y 53.9443, Z -6.3333, A 0.000, B 0.000, C 0.000 }
gfCNCPoint5[2024] = {X 326.1156, Y 54.2520, Z -6.3333, A 0.000, B 0.000, C 0.000 }
gfCNCPoint5[2025] = {X 326.9044, Y 54.7476, Z -6.3333, A 0.000, B 0.000, C 0.000 }
gfCNCPoint5[2026] = {X 327.5631, Y 55.4063, Z -6.3333, A 0.000, B 0.000, C 0.000 }
gfCNCPoint5[2027] = {X 328.0587, Y 56.1950, Z -6.3333, A 0.000, B 0.000, C 0.000 }
gfCNCPoint5[2028] = {X 328.3664, Y 57.0743, Z -6.3333, A 0.000, B 0.000, C 0.000 }
gfCNCPoint5[2029] = {X 328.4707, Y 58.0000, Z -6.3333, A 0.000, B 0.000, C 0.000 }
gfCNCPoint5[2030] = {X 328.4707, Y 58.9350, Z -6.3333, A 0.000, B 0.000, C 0.000 }
gfCNCPoint5[2031] = {X 328.3761, Y 59.7984, Z -6.3333, A 0.000, B 0.000, C 0.000 }
gfCNCPoint5[2032] = {X 328.1059, Y 60.6238, Z -6.3333, A 0.000, B 0.000, C 0.000 }
gfCNCPoint5[2033] = {X 327.6716, Y 61.3760, Z -6.3333, A 0.000, B 0.000, C 0.000 }
gfCNCPoint5[2034] = {X 327.0918, Y 62.0227, Z -6.3333, A 0.000, B 0.000, C 0.000 }
gfCNCPoint5[2035] = {X 326.3913, Y 62.5363, Z -6.3333, A 0.000, B 0.000, C 0.000 }
gfCNCPoint5[2036] = {X 325.6001, Y 62.8946, Z -6.3333, A 0.000, B 0.000, C 0.000 }
gfCNCPoint5[2037] = {X 324.7521, Y 63.0825, Z -6.3333, A 0.000, B 0.000, C 0.000 }
gfCNCPoint5[2038] = {X 324.7539, Y 83.2304, Z -6.3333, A 0.000, B 0.000, C 0.000 }
gfCNCPoint5[2039] = {X 324.7674, Y 84.6152, Z -6.3333, A 0.000, B 0.000, C 0.000 }
gfCNCPoint5[2040] = {X 324.8479, Y 85.8841, Z -6.3333, A 0.000, B 0.000, C 0.000 }
gfCNCPoint5[2041] = {X 325.0779, Y 87.1344, Z -6.3333, A 0.000, B 0.000, C 0.000 }
gfCNCPoint5[2042] = {X 325.3540, Y 87.4454, Z -6.3333, A 0.000, B 0.000, C 0.000 }
gfCNCPoint5[2043] = {X 325.6979, Y 87.6791, Z -6.3333, A 0.000, B 0.000, C 0.000 }
gfCNCPoint5[2044] = {X 326.1511, Y 87.9356, Z -6.3333, A 0.000, B 0.000, C 0.000 }
gfCNCPoint5[2045] = {X 327.6071, Y 88.5401, Z -6.3333, A 0.000, B 0.000, C 0.000 }
gfCNCPoint5[2046] = {X 329.1206, Y 88.9812, Z -6.3333, A 0.000, B 0.000, C 0.000 }
gfCNCPoint5[2047] = {X 331.4024, Y 89.4562, Z -6.3333, A 0.000, B 0.000, C 0.000 }
gfCNCPoint5[2048] = {X 333.7049, Y 89.8186, Z -6.3333, A 0.000, B 0.000, C 0.000 }
gfCNCPoint5[2049] = {X 336.0223, Y 90.0674, Z -6.3333, A 0.000, B 0.000, C 0.000 }
gfCNCPoint5[2050] = {X 340.3975, Y 90.3620, Z -6.3333, A 0.000, B 0.000, C 0.000 }
gfCNCPoint5[2051] = {X 344.7798, Y 90.5160, Z -6.3333, A 0.000, B 0.000, C 0.000 }
gfCNCPoint5[2052] = {X 349.1649, Y 90.5293, Z -6.3333, A 0.000, B 0.000, C 0.000 }
gfCNCPoint5[2053] = {X 353.3215, Y 90.4609, Z -6.3333, A 0.000, B 0.000, C 0.000 }
gfCNCPoint5[2054] = {X 357.4729, Y 90.2416, Z -6.3333, A 0.000, B 0.000, C 0.000 }
gfCNCPoint5[2055] = {X 361.6136, Y 89.8718, Z -6.3333, A 0.000, B 0.000, C 0.000 }
gfCNCPoint5[2056] = {X 363.7037, Y 89.5835, Z -6.3333, A 0.000, B 0.000, C 0.000 }
gfCNCPoint5[2057] = {X 365.7746, Y 89.1798, Z -6.3333, A 0.000, B 0.000, C 0.000 }
gfCNCPoint5[2058] = {X 367.8199, Y 88.6619, Z -6.3333, A 0.000, B 0.000, C 0.000 }
gfCNCPoint5[2059] = {X 368.7684, Y 88.3430, Z -6.3333, A 0.000, B 0.000, C 0.000 }
gfCNCPoint5[2060] = {X 369.6752, Y 87.9198, Z -6.3333, A 0.000, B 0.000, C 0.000 }
gfCNCPoint5[2061] = {X 370.5288, Y 87.3976, Z -6.3333, A 0.000, B 0.000, C 0.000 }
gfCNCPoint5[2062] = {X 370.7225, Y 87.1960, Z -6.3333, A 0.000, B 0.000, C 0.000 }
gfCNCPoint5[2063] = {X 370.8224, Y 86.9349, Z -6.3333, A 0.000, B 0.000, C 0.000 }
gfCNCPoint5[2064] = {X 371.0151, Y 85.3871, Z -6.3333, A 0.000, B 0.000, C 0.000 }
gfCNCPoint5[2065] = {X 371.0794, Y 83.8287, Z -6.3333, A 0.000, B 0.000, C 0.000 }
gfCNCPoint5[2066] = {X 371.0801, Y 63.0708, Z -6.3333, A 0.000, B 0.000, C 0.000 }
gfCNCPoint5[2067] = {X 370.9775, Y 63.0586, Z -6.3333, A 0.000, B 0.000, C 0.000 }
gfCNCPoint5[2068] = {X 370.8753, Y 63.0439, Z -6.3333, A 0.000, B 0.000, C 0.000 }
gfCNCPoint5[2069] = {X 369.9379, Y 62.7818, Z -6.3333, A 0.000, B 0.000, C 0.000 }
gfCNCPoint5[2070] = {X 369.0871, Y 62.3090, Z -6.3333, A 0.000, B 0.000, C 0.000 }
gfCNCPoint5[2071] = {X 368.3694, Y 61.6514, Z -6.3333, A 0.000, B 0.000, C 0.000 }
gfCNCPoint5[2072] = {X 367.8242, Y 60.8451, Z -6.3333, A 0.000, B 0.000, C 0.000 }
gfCNCPoint5[2073] = {X 367.4813, Y 59.9341, Z -6.3333, A 0.000, B 0.000, C 0.000 }
gfCNCPoint5[2074] = {X 367.3594, Y 58.9684, Z -6.3333, A 0.000, B 0.000, C 0.000 }
gfCNCPoint5[2075] = {X 367.3593, Y 58.0000, Z -6.3333, A 0.000, B 0.000, C 0.000 }
gfCNCPoint5[2076] = {X 367.4636, Y 57.0743, Z -6.3333, A 0.000, B 0.000, C 0.000 }
gfCNCPoint5[2077] = {X 367.7713, Y 56.1950, Z -6.3333, A 0.000, B 0.000, C 0.000 }
gfCNCPoint5[2078] = {X 368.2669, Y 55.4063, Z -6.3333, A 0.000, B 0.000, C 0.000 }
gfCNCPoint5[2079] = {X 368.9256, Y 54.7476, Z -6.3333, A 0.000, B 0.000, C 0.000 }
gfCNCPoint5[2080] = {X 369.7143, Y 54.2520, Z -6.3333, A 0.000, B 0.000, C 0.000 }
gfCNCPoint5[2081] = {X 370.5936, Y 53.9443, Z -6.3333, A 0.000, B 0.000, C 0.000 }
gfCNCPoint5[2082] = {X 371.5193, Y 53.8400, Z -6.3333, A 0.000, B 0.000, C 0.000 }
gfCNCPoint5[2083] = {X 388.0597, Y 53.8400, Z -6.3333, A 0.000, B 0.000, C 0.000 }
gfCNCPoint5[2084] = {X 388.9854, Y 53.9443, Z -6.3333, A 0.000, B 0.000, C 0.000 }
gfCNCPoint5[2085] = {X 389.8646, Y 54.2520, Z -6.3333, A 0.000, B 0.000, C 0.000 }
gfCNCPoint5[2086] = {X 390.6534, Y 54.7476, Z -6.3333, A 0.000, B 0.000, C 0.000 }
gfCNCPoint5[2087] = {X 391.3121, Y 55.4063, Z -6.3333, A 0.000, B 0.000, C 0.000 }
gfCNCPoint5[2088] = {X 391.8077, Y 56.1950, Z -6.3333, A 0.000, B 0.000, C 0.000 }
gfCNCPoint5[2089] = {X 392.1154, Y 57.0743, Z -6.3333, A 0.000, B 0.000, C 0.000 }
gfCNCPoint5[2090] = {X 392.2197, Y 58.0000, Z -6.3333, A 0.000, B 0.000, C 0.000 }
gfCNCPoint5[2091] = {X 392.2197, Y 58.9342, Z -6.3333, A 0.000, B 0.000, C 0.000 }
gfCNCPoint5[2092] = {X 392.1115, Y 59.8766, Z -6.3333, A 0.000, B 0.000, C 0.000 }
gfCNCPoint5[2093] = {X 391.7927, Y 60.7699, Z -6.3333, A 0.000, B 0.000, C 0.000 }
gfCNCPoint5[2094] = {X 391.2499, Y 61.6050, Z -6.3333, A 0.000, B 0.000, C 0.000 }
gfCNCPoint5[2095] = {X 390.5250, Y 62.2881, Z -6.3333, A 0.000, B 0.000, C 0.000 }
gfCNCPoint5[2096] = {X 389.6593, Y 62.7804, Z -6.3333, A 0.000, B 0.000, C 0.000 }
gfCNCPoint5[2097] = {X 388.7016, Y 63.0542, Z -6.3333, A 0.000, B 0.000, C 0.000 }
gfCNCPoint5[2098] = {X 388.6014, Y 63.0690, Z -6.3333, A 0.000, B 0.000, C 0.000 }
gfCNCPoint5[2099] = {X 388.5008, Y 63.0814, Z -6.3333, A 0.000, B 0.000, C 0.000 }
gfCNCPoint5[2100] = {X 388.4976, Y 84.6154, Z -6.3333, A 0.000, B 0.000, C 0.000 }
gfCNCPoint5[2101] = {X 388.4382, Y 86.2600, Z -6.3333, A 0.000, B 0.000, C 0.000 }
gfCNCPoint5[2102] = {X 388.2356, Y 87.8931, Z -6.3333, A 0.000, B 0.000, C 0.000 }
gfCNCPoint5[2103] = {X 387.8913, Y 89.5023, Z -6.3333, A 0.000, B 0.000, C 0.000 }
gfCNCPoint5[2104] = {X 387.3662, Y 91.0683, Z -6.3333, A 0.000, B 0.000, C 0.000 }
gfCNCPoint5[2105] = {X 386.6267, Y 92.5452, Z -6.3333, A 0.000, B 0.000, C 0.000 }
gfCNCPoint5[2106] = {X 385.6874, Y 93.9038, Z -6.3333, A 0.000, B 0.000, C 0.000 }
gfCNCPoint5[2107] = {X 384.5669, Y 95.1172, Z -6.3333, A 0.000, B 0.000, C 0.000 }
gfCNCPoint5[2108] = {X 383.0653, Y 96.3826, Z -6.3333, A 0.000, B 0.000, C 0.000 }
gfCNCPoint5[2109] = {X 381.4379, Y 97.4814, Z -6.3333, A 0.000, B 0.000, C 0.000 }
gfCNCPoint5[2110] = {X 379.7030, Y 98.4011, Z -6.3333, A 0.000, B 0.000, C 0.000 }
gfCNCPoint5[2111] = {X 377.4420, Y 99.3516, Z -6.3333, A 0.000, B 0.000, C 0.000 }
gfCNCPoint5[2112] = {X 375.1190, Y 100.1382, Z -6.3333, A 0.000, B 0.000, C 0.000 }
gfCNCPoint5[2113] = {X 372.7456, Y 100.7567, Z -6.3333, A 0.000, B 0.000, C 0.000 }
gfCNCPoint5[2114] = {X 368.8427, Y 101.5093, Z -6.3333, A 0.000, B 0.000, C 0.000 }
gfCNCPoint5[2115] = {X 364.9075, Y 102.0684, Z -6.3333, A 0.000, B 0.000, C 0.000 }
gfCNCPoint5[2116] = {X 360.9495, Y 102.4328, Z -6.3333, A 0.000, B 0.000, C 0.000 }
gfCNCPoint5[2117] = {X 357.0957, Y 102.6576, Z -6.3333, A 0.000, B 0.000, C 0.000 }
gfCNCPoint5[2118] = {X 353.2381, Y 102.8028, Z -6.3333, A 0.000, B 0.000, C 0.000 }
gfCNCPoint5[2119] = {X 353.3474, Y 106.8013, Z -6.3333, A 0.000, B 0.000, C 0.000 }
gfCNCPoint5[2120] = {X 353.2359, Y 102.7228, Z -6.3333, A 0.000, B 0.000, C 0.000 }
gfCNCPoint5[2121] = {X 348.1836, Y 102.7926, Z -6.3333, A 0.000, B 0.000, C 0.000 }
gfCNCPoint5[2122] = {X 343.1312, Y 102.7259, Z -6.3333, A 0.000, B 0.000, C 0.000 }
gfCNCPoint5[2123] = {X 338.0824, Y 102.5228, Z -6.3333, A 0.000, B 0.000, C 0.000 }
gfCNCPoint5[2124] = {X 334.1379, Y 102.2466, Z -6.3333, A 0.000, B 0.000, C 0.000 }
gfCNCPoint5[2125] = {X 330.2083, Y 101.8058, Z -6.3333, A 0.000, B 0.000, C 0.000 }
gfCNCPoint5[2126] = {X 326.3006, Y 101.2013, Z -6.3333, A 0.000, B 0.000, C 0.000 }
gfCNCPoint5[2127] = {X 323.4680, Y 100.6003, Z -6.3333, A 0.000, B 0.000, C 0.000 }
gfCNCPoint5[2128] = {X 320.6875, Y 99.7923, Z -6.3333, A 0.000, B 0.000, C 0.000 }
gfCNCPoint5[2129] = {X 317.9740, Y 98.7815, Z -6.3333, A 0.000, B 0.000, C 0.000 }
gfCNCPoint5[2130] = {X 316.4792, Y 98.0921, Z -6.3333, A 0.000, B 0.000, C 0.000 }
gfCNCPoint5[2131] = {X 315.0473, Y 97.2801, Z -6.3333, A 0.000, B 0.000, C 0.000 }
gfCNCPoint5[2132] = {X 313.6883, Y 96.3513, Z -6.3333, A 0.000, B 0.000, C 0.000 }
gfCNCPoint5[2133] = {X 312.4117, Y 95.3120, Z -6.3333, A 0.000, B 0.000, C 0.000 }
gfCNCPoint5[2134] = {X 311.4281, Y 94.3334, Z -6.3333, A 0.000, B 0.000, C 0.000 }
gfCNCPoint5[2135] = {X 310.5674, Y 93.2451, Z -6.3333, A 0.000, B 0.000, C 0.000 }
gfCNCPoint5[2136] = {X 309.8417, Y 92.0626, Z -6.3333, A 0.000, B 0.000, C 0.000 }
gfCNCPoint5[2137] = {X 309.2613, Y 90.8023, Z -6.3333, A 0.000, B 0.000, C 0.000 }
gfCNCPoint5[2138] = {X 308.8343, Y 89.4822, Z -6.3333, A 0.000, B 0.000, C 0.000 }
gfCNCPoint5[2139] = {X 308.4951, Y 87.8792, Z -6.3333, A 0.000, B 0.000, C 0.000 }
gfCNCPoint5[2140] = {X 308.2948, Y 86.2530, Z -6.3333, A 0.000, B 0.000, C 0.000 }
gfCNCPoint5[2141] = {X 308.2347, Y 84.6156, Z -6.3333, A 0.000, B 0.000, C 0.000 }
gfCNCPoint5[2142] = {X 308.2360, Y 62.9981, Z -6.3333, A 0.000, B 0.000, C 0.000 }
gfCNCPoint5[2143] = {X 307.3944, Y 62.8330, Z -6.3333, A 0.000, B 0.000, C 0.000 }
gfCNCPoint5[2144] = {X 306.6059, Y 62.4957, Z -6.3333, A 0.000, B 0.000, C 0.000 }
gfCNCPoint5[2145] = {X 305.9054, Y 62.0009, Z -6.3333, A 0.000, B 0.000, C 0.000 }
gfCNCPoint5[2146] = {X 305.3237, Y 61.3707, Z -6.3333, A 0.000, B 0.000, C 0.000 }
gfCNCPoint5[2147] = {X 304.8867, Y 60.6328, Z -6.3333, A 0.000, B 0.000, C 0.000 }
gfCNCPoint5[2148] = {X 304.6135, Y 59.8199, Z -6.3333, A 0.000, B 0.000, C 0.000 }
gfCNCPoint5[2149] = {X 304.5164, Y 58.9678, Z -6.3333, A 0.000, B 0.000, C 0.000 }
gfCNCPoint5[2150] = {X 304.5162, Y 58.0000, Z -6.3333, A 0.000, B 0.000, C 0.000 }
gfCNCPoint5[2151] = {X 304.6185, Y 57.0921, Z -6.3333, A 0.000, B 0.000, C 0.000 }
gfCNCPoint5[2152] = {X 304.9203, Y 56.2298, Z -6.3333, A 0.000, B 0.000, C 0.000 }
gfCNCPoint5[2153] = {X 305.4064, Y 55.4562, Z -6.3333, A 0.000, B 0.000, C 0.000 }
gfCNCPoint5[2154] = {X 306.0524, Y 54.8101, Z -6.3333, A 0.000, B 0.000, C 0.000 }
gfCNCPoint5[2155] = {X 306.8260, Y 54.3240, Z -6.3333, A 0.000, B 0.000, C 0.000 }
gfCNCPoint5[2156] = {X 307.6883, Y 54.0223, Z -6.3333, A 0.000, B 0.000, C 0.000 }
gfCNCPoint5[2157] = {X 308.5962, Y 53.9200, Z -6.3333, A 0.000, B 0.000, C 0.000 }
gfCNCPoint5[2158] = {X 324.3107, Y 53.9200, Z -6.3333, A 0.000, B 0.000, C 0.000 }
gfCNCPoint5[2159] = {X 325.2186, Y 54.0223, Z -6.3333, A 0.000, B 0.000, C 0.000 }
gfCNCPoint5[2160] = {X 326.0809, Y 54.3240, Z -6.3333, A 0.000, B 0.000, C 0.000 }
gfCNCPoint5[2161] = {X 326.8545, Y 54.8101, Z -6.3333, A 0.000, B 0.000, C 0.000 }
gfCNCPoint5[2162] = {X 327.5006, Y 55.4562, Z -6.3333, A 0.000, B 0.000, C 0.000 }
gfCNCPoint5[2163] = {X 327.9866, Y 56.2298, Z -6.3333, A 0.000, B 0.000, C 0.000 }
gfCNCPoint5[2164] = {X 328.2884, Y 57.0921, Z -6.3333, A 0.000, B 0.000, C 0.000 }
gfCNCPoint5[2165] = {X 328.3907, Y 58.0000, Z -6.3333, A 0.000, B 0.000, C 0.000 }
gfCNCPoint5[2166] = {X 328.3907, Y 58.9345, Z -6.3333, A 0.000, B 0.000, C 0.000 }
gfCNCPoint5[2167] = {X 328.2958, Y 59.7914, Z -6.3333, A 0.000, B 0.000, C 0.000 }
gfCNCPoint5[2168] = {X 328.0245, Y 60.6098, Z -6.3333, A 0.000, B 0.000, C 0.000 }
gfCNCPoint5[2169] = {X 327.5888, Y 61.3537, Z -6.3333, A 0.000, B 0.000, C 0.000 }
gfCNCPoint5[2170] = {X 327.0077, Y 61.9906, Z -6.3333, A 0.000, B 0.000, C 0.000 }
gfCNCPoint5[2171] = {X 326.3068, Y 62.4926, Z -6.3333, A 0.000, B 0.000, C 0.000 }
gfCNCPoint5[2172] = {X 325.5167, Y 62.8376, Z -6.3333, A 0.000, B 0.000, C 0.000 }
gfCNCPoint5[2173] = {X 324.6721, Y 63.0105, Z -6.3333, A 0.000, B 0.000, C 0.000 }
gfCNCPoint5[2174] = {X 324.6739, Y 83.2308, Z -6.3333, A 0.000, B 0.000, C 0.000 }
gfCNCPoint5[2175] = {X 324.6874, Y 84.6156, Z -6.3333, A 0.000, B 0.000, C 0.000 }
gfCNCPoint5[2176] = {X 324.7694, Y 85.9010, Z -6.3333, A 0.000, B 0.000, C 0.000 }
gfCNCPoint5[2177] = {X 325.0037, Y 87.1676, Z -6.3333, A 0.000, B 0.000, C 0.000 }
gfCNCPoint5[2178] = {X 325.2950, Y 87.5001, Z -6.3333, A 0.000, B 0.000, C 0.000 }
gfCNCPoint5[2179] = {X 325.6599, Y 87.7496, Z -6.3333, A 0.000, B 0.000, C 0.000 }
gfCNCPoint5[2180] = {X 326.1140, Y 88.0066, Z -6.3333, A 0.000, B 0.000, C 0.000 }
gfCNCPoint5[2181] = {X 327.5793, Y 88.6151, Z -6.3333, A 0.000, B 0.000, C 0.000 }
gfCNCPoint5[2182] = {X 329.1025, Y 89.0591, Z -6.3333, A 0.000, B 0.000, C 0.000 }
gfCNCPoint5[2183] = {X 331.3881, Y 89.5349, Z -6.3333, A 0.000, B 0.000, C 0.000 }
gfCNCPoint5[2184] = {X 333.6944, Y 89.8979, Z -6.3333, A 0.000, B 0.000, C 0.000 }
gfCNCPoint5[2185] = {X 336.0157, Y 90.1471, Z -6.3333, A 0.000, B 0.000, C 0.000 }
gfCNCPoint5[2186] = {X 340.3934, Y 90.4419, Z -6.3333, A 0.000, B 0.000, C 0.000 }
gfCNCPoint5[2187] = {X 344.7783, Y 90.5960, Z -6.3333, A 0.000, B 0.000, C 0.000 }
gfCNCPoint5[2188] = {X 349.1659, Y 90.6093, Z -6.3333, A 0.000, B 0.000, C 0.000 }
gfCNCPoint5[2189] = {X 353.3251, Y 90.5408, Z -6.3333, A 0.000, B 0.000, C 0.000 }
gfCNCPoint5[2190] = {X 357.4791, Y 90.3213, Z -6.3333, A 0.000, B 0.000, C 0.000 }
gfCNCPoint5[2191] = {X 361.6223, Y 89.9513, Z -6.3333, A 0.000, B 0.000, C 0.000 }
gfCNCPoint5[2192] = {X 363.7168, Y 89.6624, Z -6.3333, A 0.000, B 0.000, C 0.000 }
gfCNCPoint5[2193] = {X 365.7920, Y 89.2578, Z -6.3333, A 0.000, B 0.000, C 0.000 }
gfCNCPoint5[2194] = {X 367.8417, Y 88.7389, Z -6.3333, A 0.000, B 0.000, C 0.000 }
gfCNCPoint5[2195] = {X 368.7985, Y 88.4171, Z -6.3333, A 0.000, B 0.000, C 0.000 }
gfCNCPoint5[2196] = {X 369.7132, Y 87.9902, Z -6.3333, A 0.000, B 0.000, C 0.000 }
gfCNCPoint5[2197] = {X 370.5743, Y 87.4634, Z -6.3333, A 0.000, B 0.000, C 0.000 }
gfCNCPoint5[2198] = {X 370.7901, Y 87.2389, Z -6.3333, A 0.000, B 0.000, C 0.000 }
gfCNCPoint5[2199] = {X 370.9013, Y 86.9481, Z -6.3333, A 0.000, B 0.000, C 0.000 }
gfCNCPoint5[2200] = {X 371.0948, Y 85.3937, Z -6.3333, A 0.000, B 0.000, C 0.000 }
gfCNCPoint5[2201] = {X 371.1594, Y 83.8286, Z -6.3333, A 0.000, B 0.000, C 0.000 }
gfCNCPoint5[2202] = {X 371.1601, Y 62.9982, Z -6.3333, A 0.000, B 0.000, C 0.000 }
gfCNCPoint5[2203] = {X 371.0236, Y 62.9838, Z -6.3333, A 0.000, B 0.000, C 0.000 }
gfCNCPoint5[2204] = {X 370.8877, Y 62.9649, Z -6.3333, A 0.000, B 0.000, C 0.000 }
gfCNCPoint5[2205] = {X 369.9683, Y 62.7078, Z -6.3333, A 0.000, B 0.000, C 0.000 }
gfCNCPoint5[2206] = {X 369.1338, Y 62.2441, Z -6.3333, A 0.000, B 0.000, C 0.000 }
gfCNCPoint5[2207] = {X 368.4300, Y 61.5991, Z -6.3333, A 0.000, B 0.000, C 0.000 }
gfCNCPoint5[2208] = {X 367.8953, Y 60.8083, Z -6.3333, A 0.000, B 0.000, C 0.000 }
gfCNCPoint5[2209] = {X 367.5589, Y 59.9149, Z -6.3333, A 0.000, B 0.000, C 0.000 }
gfCNCPoint5[2210] = {X 367.4394, Y 58.9678, Z -6.3333, A 0.000, B 0.000, C 0.000 }
gfCNCPoint5[2211] = {X 367.4393, Y 58.0000, Z -6.3333, A 0.000, B 0.000, C 0.000 }
gfCNCPoint5[2212] = {X 367.5416, Y 57.0921, Z -6.3333, A 0.000, B 0.000, C 0.000 }
gfCNCPoint5[2213] = {X 367.8433, Y 56.2298, Z -6.3333, A 0.000, B 0.000, C 0.000 }
gfCNCPoint5[2214] = {X 368.3294, Y 55.4562, Z -6.3333, A 0.000, B 0.000, C 0.000 }
gfCNCPoint5[2215] = {X 368.9754, Y 54.8101, Z -6.3333, A 0.000, B 0.000, C 0.000 }
gfCNCPoint5[2216] = {X 369.7490, Y 54.3240, Z -6.3333, A 0.000, B 0.000, C 0.000 }
gfCNCPoint5[2217] = {X 370.6114, Y 54.0223, Z -6.3333, A 0.000, B 0.000, C 0.000 }
gfCNCPoint5[2218] = {X 371.5193, Y 53.9200, Z -6.3333, A 0.000, B 0.000, C 0.000 }
gfCNCPoint5[2219] = {X 388.0597, Y 53.9200, Z -6.3333, A 0.000, B 0.000, C 0.000 }
gfCNCPoint5[2220] = {X 388.9676, Y 54.0223, Z -6.3333, A 0.000, B 0.000, C 0.000 }
gfCNCPoint5[2221] = {X 389.8299, Y 54.3240, Z -6.3333, A 0.000, B 0.000, C 0.000 }
gfCNCPoint5[2222] = {X 390.6035, Y 54.8101, Z -6.3333, A 0.000, B 0.000, C 0.000 }
gfCNCPoint5[2223] = {X 391.2496, Y 55.4562, Z -6.3333, A 0.000, B 0.000, C 0.000 }
gfCNCPoint5[2224] = {X 391.7356, Y 56.2298, Z -6.3333, A 0.000, B 0.000, C 0.000 }
gfCNCPoint5[2225] = {X 392.0374, Y 57.0921, Z -6.3333, A 0.000, B 0.000, C 0.000 }
gfCNCPoint5[2226] = {X 392.1397, Y 58.0000, Z -6.3333, A 0.000, B 0.000, C 0.000 }
gfCNCPoint5[2227] = {X 392.1397, Y 58.9342, Z -6.3333, A 0.000, B 0.000, C 0.000 }
gfCNCPoint5[2228] = {X 392.0336, Y 59.8584, Z -6.3333, A 0.000, B 0.000, C 0.000 }
gfCNCPoint5[2229] = {X 391.7209, Y 60.7346, Z -6.3333, A 0.000, B 0.000, C 0.000 }
gfCNCPoint5[2230] = {X 391.1885, Y 61.5537, Z -6.3333, A 0.000, B 0.000, C 0.000 }
gfCNCPoint5[2231] = {X 390.4775, Y 62.2237, Z -6.3333, A 0.000, B 0.000, C 0.000 }
gfCNCPoint5[2232] = {X 389.6283, Y 62.7067, Z -6.3333, A 0.000, B 0.000, C 0.000 }
gfCNCPoint5[2233] = {X 388.6889, Y 62.9752, Z -6.3333, A 0.000, B 0.000, C 0.000 }
gfCNCPoint5[2234] = {X 388.5557, Y 62.9943, Z -6.3333, A 0.000, B 0.000, C 0.000 }
gfCNCPoint5[2235] = {X 388.4219, Y 63.0091, Z -6.3333, A 0.000, B 0.000, C 0.000 }
gfCNCPoint5[2236] = {X 388.4196, Y 63.1547, Z -6.3333, A 0.000, B 0.000, C 0.000 }
gfCNCPoint5[2237] = {X 388.4176, Y 84.6157, Z -6.3333, A 0.000, B 0.000, C 0.000 }
gfCNCPoint5[2238] = {X 388.3585, Y 86.2534, Z -6.3333, A 0.000, B 0.000, C 0.000 }
gfCNCPoint5[2239] = {X 388.1567, Y 87.8797, Z -6.3333, A 0.000, B 0.000, C 0.000 }
gfCNCPoint5[2240] = {X 387.8139, Y 89.4822, Z -6.3333, A 0.000, B 0.000, C 0.000 }
gfCNCPoint5[2241] = {X 387.2923, Y 91.0376, Z -6.3333, A 0.000, B 0.000, C 0.000 }
gfCNCPoint5[2242] = {X 386.5579, Y 92.5044, Z -6.3333, A 0.000, B 0.000, C 0.000 }
gfCNCPoint5[2243] = {X 385.6250, Y 93.8537, Z -6.3333, A 0.000, B 0.000, C 0.000 }
gfCNCPoint5[2244] = {X 384.5121, Y 95.0589, Z -6.3333, A 0.000, B 0.000, C 0.000 }
gfCNCPoint5[2245] = {X 383.0171, Y 96.3188, Z -6.3333, A 0.000, B 0.000, C 0.000 }
gfCNCPoint5[2246] = {X 381.3967, Y 97.4128, Z -6.3333, A 0.000, B 0.000, C 0.000 }
gfCNCPoint5[2247] = {X 379.6693, Y 98.3285, Z -6.3333, A 0.000, B 0.000, C 0.000 }
gfCNCPoint5[2248] = {X 377.4137, Y 99.2768, Z -6.3333, A 0.000, B 0.000, C 0.000 }
gfCNCPoint5[2249] = {X 375.0960, Y 100.0615, Z -6.3333, A 0.000, B 0.000, C 0.000 }
gfCNCPoint5[2250] = {X 372.7282, Y 100.6786, Z -6.3333, A 0.000, B 0.000, C 0.000 }
gfCNCPoint5[2251] = {X 368.8293, Y 101.4304, Z -6.3333, A 0.000, B 0.000, C 0.000 }
gfCNCPoint5[2252] = {X 364.8980, Y 101.9890, Z -6.3333, A 0.000, B 0.000, C 0.000 }
gfCNCPoint5[2253] = {X 360.9440, Y 102.3530, Z -6.3333, A 0.000, B 0.000, C 0.000 }
gfCNCPoint5[2254] = {X 357.0919, Y 102.5777, Z -6.3333, A 0.000, B 0.000, C 0.000 }
gfCNCPoint5[2255] = {X 353.2359, Y 102.7228, Z -6.3333, A 0.000, B 0.000, C 0.000 }
gfCNCPoint5[2256] = {X 353.3452, Y 106.7213, Z -6.3333, A 0.000, B 0.000, C 0.000 }
gfCNCPoint5[2257] = {X 353.2338, Y 102.6429, Z -6.3333, A 0.000, B 0.000, C 0.000 }
gfCNCPoint5[2258] = {X 348.1835, Y 102.7126, Z -6.3333, A 0.000, B 0.000, C 0.000 }
gfCNCPoint5[2259] = {X 343.1332, Y 102.6459, Z -6.3333, A 0.000, B 0.000, C 0.000 }
gfCNCPoint5[2260] = {X 338.0866, Y 102.4429, Z -6.3333, A 0.000, B 0.000, C 0.000 }
gfCNCPoint5[2261] = {X 334.1453, Y 102.1669, Z -6.3333, A 0.000, B 0.000, C 0.000 }
gfCNCPoint5[2262] = {X 330.2189, Y 101.7265, Z -6.3333, A 0.000, B 0.000, C 0.000 }
gfCNCPoint5[2263] = {X 326.3144, Y 101.1225, Z -6.3333, A 0.000, B 0.000, C 0.000 }
gfCNCPoint5[2264] = {X 323.4875, Y 100.5227, Z -6.3333, A 0.000, B 0.000, C 0.000 }
gfCNCPoint5[2265] = {X 320.7126, Y 99.7163, Z -6.3333, A 0.000, B 0.000, C 0.000 }
gfCNCPoint5[2266] = {X 318.0046, Y 98.7076, Z -6.3333, A 0.000, B 0.000, C 0.000 }
gfCNCPoint5[2267] = {X 316.5158, Y 98.0210, Z -6.3333, A 0.000, B 0.000, C 0.000 }
gfCNCPoint5[2268] = {X 315.0897, Y 97.2123, Z -6.3333, A 0.000, B 0.000, C 0.000 }
gfCNCPoint5[2269] = {X 313.7361, Y 96.2872, Z -6.3333, A 0.000, B 0.000, C 0.000 }
gfCNCPoint5[2270] = {X 312.4647, Y 95.2521, Z -6.3333, A 0.000, B 0.000, C 0.000 }
gfCNCPoint5[2271] = {X 311.4878, Y 94.2802, Z -6.3333, A 0.000, B 0.000, C 0.000 }
gfCNCPoint5[2272] = {X 310.6330, Y 93.1994, Z -6.3333, A 0.000, B 0.000, C 0.000 }
gfCNCPoint5[2273] = {X 309.9123, Y 92.0249, Z -6.3333, A 0.000, B 0.000, C 0.000 }
gfCNCPoint5[2274] = {X 309.3358, Y 90.7732, Z -6.3333, A 0.000, B 0.000, C 0.000 }
gfCNCPoint5[2275] = {X 308.9118, Y 89.4621, Z -6.3333, A 0.000, B 0.000, C 0.000 }
gfCNCPoint5[2276] = {X 308.5740, Y 87.8658, Z -6.3333, A 0.000, B 0.000, C 0.000 }
gfCNCPoint5[2277] = {X 308.3745, Y 86.2464, Z -6.3333, A 0.000, B 0.000, C 0.000 }
gfCNCPoint5[2278] = {X 308.3147, Y 84.6159, Z -6.3333, A 0.000, B 0.000, C 0.000 }
gfCNCPoint5[2279] = {X 308.3160, Y 62.9242, Z -6.3333, A 0.000, B 0.000, C 0.000 }
gfCNCPoint5[2280] = {X 307.4735, Y 62.7733, Z -6.3333, A 0.000, B 0.000, C 0.000 }
gfCNCPoint5[2281] = {X 306.6824, Y 62.4465, Z -6.3333, A 0.000, B 0.000, C 0.000 }
gfCNCPoint5[2282] = {X 305.9790, Y 61.9590, Z -6.3333, A 0.000, B 0.000, C 0.000 }
gfCNCPoint5[2283] = {X 305.3954, Y 61.3329, Z -6.3333, A 0.000, B 0.000, C 0.000 }
gfCNCPoint5[2284] = {X 304.9583, Y 60.5970, Z -6.3333, A 0.000, B 0.000, C 0.000 }
gfCNCPoint5[2285] = {X 304.6878, Y 59.7850, Z -6.3333, A 0.000, B 0.000, C 0.000 }
gfCNCPoint5[2286] = {X 304.5962, Y 58.9341, Z -6.3333, A 0.000, B 0.000, C 0.000 }
gfCNCPoint5[2287] = {X 304.5962, Y 58.0000, Z -6.3333, A 0.000, B 0.000, C 0.000 }
gfCNCPoint5[2288] = {X 304.6965, Y 57.1099, Z -6.3333, A 0.000, B 0.000, C 0.000 }
gfCNCPoint5[2289] = {X 304.9923, Y 56.2645, Z -6.3333, A 0.000, B 0.000, C 0.000 }
gfCNCPoint5[2290] = {X 305.4689, Y 55.5060, Z -6.3333, A 0.000, B 0.000, C 0.000 }
gfCNCPoint5[2291] = {X 306.1023, Y 54.8727, Z -6.3333, A 0.000, B 0.000, C 0.000 }
gfCNCPoint5[2292] = {X 306.8607, Y 54.3961, Z -6.3333, A 0.000, B 0.000, C 0.000 }
gfCNCPoint5[2293] = {X 307.7061, Y 54.1003, Z -6.3333, A 0.000, B 0.000, C 0.000 }
gfCNCPoint5[2294] = {X 308.5962, Y 54.0000, Z -6.3333, A 0.000, B 0.000, C 0.000 }
gfCNCPoint5[2295] = {X 324.3107, Y 54.0000, Z -6.3333, A 0.000, B 0.000, C 0.000 }
gfCNCPoint5[2296] = {X 325.2008, Y 54.1003, Z -6.3333, A 0.000, B 0.000, C 0.000 }
gfCNCPoint5[2297] = {X 326.0462, Y 54.3961, Z -6.3333, A 0.000, B 0.000, C 0.000 }
gfCNCPoint5[2298] = {X 326.8046, Y 54.8727, Z -6.3333, A 0.000, B 0.000, C 0.000 }
gfCNCPoint5[2299] = {X 327.4380, Y 55.5060, Z -6.3333, A 0.000, B 0.000, C 0.000 }
gfCNCPoint5[2300] = {X 327.9146, Y 56.2645, Z -6.3333, A 0.000, B 0.000, C 0.000 }
gfCNCPoint5[2301] = {X 328.2104, Y 57.1099, Z -6.3333, A 0.000, B 0.000, C 0.000 }
gfCNCPoint5[2302] = {X 328.3107, Y 58.0000, Z -6.3333, A 0.000, B 0.000, C 0.000 }
gfCNCPoint5[2303] = {X 328.3107, Y 58.9341, Z -6.3333, A 0.000, B 0.000, C 0.000 }
gfCNCPoint5[2304] = {X 328.2154, Y 59.7845, Z -6.3333, A 0.000, B 0.000, C 0.000 }
gfCNCPoint5[2305] = {X 327.9431, Y 60.5957, Z -6.3333, A 0.000, B 0.000, C 0.000 }
gfCNCPoint5[2306] = {X 327.5059, Y 61.3313, Z -6.3333, A 0.000, B 0.000, C 0.000 }
gfCNCPoint5[2307] = {X 326.9235, Y 61.9582, Z -6.3333, A 0.000, B 0.000, C 0.000 }
gfCNCPoint5[2308] = {X 326.2221, Y 62.4483, Z -6.3333, A 0.000, B 0.000, C 0.000 }
gfCNCPoint5[2309] = {X 325.4331, Y 62.7797, Z -6.3333, A 0.000, B 0.000, C 0.000 }
gfCNCPoint5[2310] = {X 324.5920, Y 62.9373, Z -6.3333, A 0.000, B 0.000, C 0.000 }
gfCNCPoint5[2311] = {X 324.5939, Y 83.2313, Z -6.3333, A 0.000, B 0.000, C 0.000 }
gfCNCPoint5[2312] = {X 324.6074, Y 84.6159, Z -6.3333, A 0.000, B 0.000, C 0.000 }
gfCNCPoint5[2313] = {X 324.6909, Y 85.9178, Z -6.3333, A 0.000, B 0.000, C 0.000 }
gfCNCPoint5[2314] = {X 324.9294, Y 87.2004, Z -6.3333, A 0.000, B 0.000, C 0.000 }
gfCNCPoint5[2315] = {X 325.2359, Y 87.5546, Z -6.3333, A 0.000, B 0.000, C 0.000 }
gfCNCPoint5[2316] = {X 325.6219, Y 87.8200, Z -6.3333, A 0.000, B 0.000, C 0.000 }
gfCNCPoint5[2317] = {X 326.0769, Y 88.0775, Z -6.3333, A 0.000, B 0.000, C 0.000 }
gfCNCPoint5[2318] = {X 327.5515, Y 88.6901, Z -6.3333, A 0.000, B 0.000, C 0.000 }
gfCNCPoint5[2319] = {X 329.0843, Y 89.1370, Z -6.3333, A 0.000, B 0.000, C 0.000 }
gfCNCPoint5[2320] = {X 331.3738, Y 89.6136, Z -6.3333, A 0.000, B 0.000, C 0.000 }
gfCNCPoint5[2321] = {X 333.6840, Y 89.9772, Z -6.3333, A 0.000, B 0.000, C 0.000 }
gfCNCPoint5[2322] = {X 336.0092, Y 90.2269, Z -6.3333, A 0.000, B 0.000, C 0.000 }
gfCNCPoint5[2323] = {X 340.3892, Y 90.5218, Z -6.3333, A 0.000, B 0.000, C 0.000 }
gfCNCPoint5[2324] = {X 344.7764, Y 90.6760, Z -6.3333, A 0.000, B 0.000, C 0.000 }
gfCNCPoint5[2325] = {X 349.1664, Y 90.6893, Z -6.3333, A 0.000, B 0.000, C 0.000 }
gfCNCPoint5[2326] = {X 353.3283, Y 90.6207, Z -6.3333, A 0.000, B 0.000, C 0.000 }
gfCNCPoint5[2327] = {X 357.4851, Y 90.4011, Z -6.3333, A 0.000, B 0.000, C 0.000 }
gfCNCPoint5[2328] = {X 361.6311, Y 90.0308, Z -6.3333, A 0.000, B 0.000, C 0.000 }
gfCNCPoint5[2329] = {X 363.7299, Y 89.7413, Z -6.3333, A 0.000, B 0.000, C 0.000 }
gfCNCPoint5[2330] = {X 365.8095, Y 89.3359, Z -6.3333, A 0.000, B 0.000, C 0.000 }
gfCNCPoint5[2331] = {X 367.8634, Y 88.8159, Z -6.3333, A 0.000, B 0.000, C 0.000 }
gfCNCPoint5[2332] = {X 368.8286, Y 88.4913, Z -6.3333, A 0.000, B 0.000, C 0.000 }
gfCNCPoint5[2333] = {X 369.7512, Y 88.0606, Z -6.3333, A 0.000, B 0.000, C 0.000 }
gfCNCPoint5[2334] = {X 370.6198, Y 87.5292, Z -6.3333, A 0.000, B 0.000, C 0.000 }
gfCNCPoint5[2335] = {X 370.8576, Y 87.2817, Z -6.3333, A 0.000, B 0.000, C 0.000 }
gfCNCPoint5[2336] = {X 370.9802, Y 86.9612, Z -6.3333, A 0.000, B 0.000, C 0.000 }
gfCNCPoint5[2337] = {X 371.1745, Y 85.4003, Z -6.3333, A 0.000, B 0.000, C 0.000 }
gfCNCPoint5[2338] = {X 371.2394, Y 83.8286, Z -6.3333, A 0.000, B 0.000, C 0.000 }
gfCNCPoint5[2339] = {X 371.2381, Y 63.0396, Z -6.3333, A 0.000, B 0.000, C 0.000 }
gfCNCPoint5[2340] = {X 371.2440, Y 62.9246, Z -6.3333, A 0.000, B 0.000, C 0.000 }
gfCNCPoint5[2341] = {X 371.0716, Y 62.9089, Z -6.3333, A 0.000, B 0.000, C 0.000 }
gfCNCPoint5[2342] = {X 370.9001, Y 62.8858, Z -6.3333, A 0.000, B 0.000, C 0.000 }
gfCNCPoint5[2343] = {X 369.9936, Y 62.6317, Z -6.3333, A 0.000, B 0.000, C 0.000 }
gfCNCPoint5[2344] = {X 369.1717, Y 62.1727, Z -6.3333, A 0.000, B 0.000, C 0.000 }
gfCNCPoint5[2345] = {X 368.4798, Y 61.5344, Z -6.3333, A 0.000, B 0.000, C 0.000 }
gfCNCPoint5[2346] = {X 367.9563, Y 60.7520, Z -6.3333, A 0.000, B 0.000, C 0.000 }
gfCNCPoint5[2347] = {X 367.6301, Y 59.8689, Z -6.3333, A 0.000, B 0.000, C 0.000 }
gfCNCPoint5[2348] = {X 367.5193, Y 58.9341, Z -6.3333, A 0.000, B 0.000, C 0.000 }
gfCNCPoint5[2349] = {X 367.5193, Y 58.0000, Z -6.3333, A 0.000, B 0.000, C 0.000 }
gfCNCPoint5[2350] = {X 367.6196, Y 57.1099, Z -6.3333, A 0.000, B 0.000, C 0.000 }
gfCNCPoint5[2351] = {X 367.9154, Y 56.2645, Z -6.3333, A 0.000, B 0.000, C 0.000 }
gfCNCPoint5[2352] = {X 368.3920, Y 55.5060, Z -6.3333, A 0.000, B 0.000, C 0.000 }
gfCNCPoint5[2353] = {X 369.0253, Y 54.8727, Z -6.3333, A 0.000, B 0.000, C 0.000 }
gfCNCPoint5[2354] = {X 369.7837, Y 54.3961, Z -6.3333, A 0.000, B 0.000, C 0.000 }
gfCNCPoint5[2355] = {X 370.6292, Y 54.1003, Z -6.3333, A 0.000, B 0.000, C 0.000 }
gfCNCPoint5[2356] = {X 371.5193, Y 54.0000, Z -6.3333, A 0.000, B 0.000, C 0.000 }
gfCNCPoint5[2357] = {X 388.0597, Y 54.0000, Z -6.3333, A 0.000, B 0.000, C 0.000 }
gfCNCPoint5[2358] = {X 388.9498, Y 54.1003, Z -6.3333, A 0.000, B 0.000, C 0.000 }
gfCNCPoint5[2359] = {X 389.7952, Y 54.3961, Z -6.3333, A 0.000, B 0.000, C 0.000 }
gfCNCPoint5[2360] = {X 390.5536, Y 54.8727, Z -6.3333, A 0.000, B 0.000, C 0.000 }
gfCNCPoint5[2361] = {X 391.1870, Y 55.5060, Z -6.3333, A 0.000, B 0.000, C 0.000 }
gfCNCPoint5[2362] = {X 391.6636, Y 56.2645, Z -6.3333, A 0.000, B 0.000, C 0.000 }
gfCNCPoint5[2363] = {X 391.9594, Y 57.1099, Z -6.3333, A 0.000, B 0.000, C 0.000 }
gfCNCPoint5[2364] = {X 392.0597, Y 58.0000, Z -6.3333, A 0.000, B 0.000, C 0.000 }
gfCNCPoint5[2365] = {X 392.0595, Y 58.9671, Z -6.3333, A 0.000, B 0.000, C 0.000 }
gfCNCPoint5[2366] = {X 391.9519, Y 59.8563, Z -6.3333, A 0.000, B 0.000, C 0.000 }
gfCNCPoint5[2367] = {X 391.6491, Y 60.6993, Z -6.3333, A 0.000, B 0.000, C 0.000 }
gfCNCPoint5[2368] = {X 391.1271, Y 61.5024, Z -6.3333, A 0.000, B 0.000, C 0.000 }
gfCNCPoint5[2369] = {X 390.4299, Y 62.1594, Z -6.3333, A 0.000, B 0.000, C 0.000 }
gfCNCPoint5[2370] = {X 389.5973, Y 62.6329, Z -6.3333, A 0.000, B 0.000, C 0.000 }
gfCNCPoint5[2371] = {X 388.6763, Y 62.8962, Z -6.3333, A 0.000, B 0.000, C 0.000 }
gfCNCPoint5[2372] = {X 388.5100, Y 62.9193, Z -6.3333, A 0.000, B 0.000, C 0.000 }
gfCNCPoint5[2373] = {X 388.3430, Y 62.9355, Z -6.3333, A 0.000, B 0.000, C 0.000 }
gfCNCPoint5[2374] = {X 388.3396, Y 63.1540, Z -6.3333, A 0.000, B 0.000, C 0.000 }
gfCNCPoint5[2375] = {X 388.3396, Y 83.9236, Z -6.3333, A 0.000, B 0.000, C 0.000 }
gfCNCPoint5[2376] = {X 388.3376, Y 84.6159, Z -6.3333, A 0.000, B 0.000, C 0.000 }
gfCNCPoint5[2377] = {X 388.2788, Y 86.2468, Z -6.3333, A 0.000, B 0.000, C 0.000 }
gfCNCPoint5[2378] = {X 388.0779, Y 87.8663, Z -6.3333, A 0.000, B 0.000, C 0.000 }
gfCNCPoint5[2379] = {X 387.7364, Y 89.4621, Z -6.3333, A 0.000, B 0.000, C 0.000 }
gfCNCPoint5[2380] = {X 387.2185, Y 91.0068, Z -6.3333, A 0.000, B 0.000, C 0.000 }
gfCNCPoint5[2381] = {X 386.4891, Y 92.4636, Z -6.3333, A 0.000, B 0.000, C 0.000 }
gfCNCPoint5[2382] = {X 385.5625, Y 93.8037, Z -6.3333, A 0.000, B 0.000, C 0.000 }
gfCNCPoint5[2383] = {X 384.4573, Y 95.0007, Z -6.3333, A 0.000, B 0.000, C 0.000 }
gfCNCPoint5[2384] = {X 382.9688, Y 96.2550, Z -6.3333, A 0.000, B 0.000, C 0.000 }
gfCNCPoint5[2385] = {X 381.3555, Y 97.3442, Z -6.3333, A 0.000, B 0.000, C 0.000 }
gfCNCPoint5[2386] = {X 379.6357, Y 98.2560, Z -6.3333, A 0.000, B 0.000, C 0.000 }
gfCNCPoint5[2387] = {X 377.3853, Y 99.2020, Z -6.3333, A 0.000, B 0.000, C 0.000 }
gfCNCPoint5[2388] = {X 375.0731, Y 99.9849, Z -6.3333, A 0.000, B 0.000, C 0.000 }
gfCNCPoint5[2389] = {X 372.7108, Y 100.6006, Z -6.3333, A 0.000, B 0.000, C 0.000 }
gfCNCPoint5[2390] = {X 368.8159, Y 101.3516, Z -6.3333, A 0.000, B 0.000, C 0.000 }
gfCNCPoint5[2391] = {X 364.8886, Y 101.9096, Z -6.3333, A 0.000, B 0.000, C 0.000 }
gfCNCPoint5[2392] = {X 360.9386, Y 102.2732, Z -6.3333, A 0.000, B 0.000, C 0.000 }
gfCNCPoint5[2393] = {X 357.0881, Y 102.4978, Z -6.3333, A 0.000, B 0.000, C 0.000 }
gfCNCPoint5[2394] = {X 353.2338, Y 102.6429, Z -6.3333, A 0.000, B 0.000, C 0.000 }
gfCNCPoint5[2395] = {X 353.3452, Y 106.7213, Z -6.3333, A 0.000, B 0.000, C 0.000 }
gfCNCPoint5[2396] = {X 353.3452, Y 106.7213, Z -3.3333, A 0.000, B 0.000, C 0.000 }
gfCNCPoint5[2397] = {X 353.3452, Y 106.7213, Z 11.0000, A 0.000, B 0.000, C 0.000 }
gfCNCPoint5[2398] = {X 411.5985, Y 79.5924, Z 11.0000, A 0.000, B 0.000, C 0.000 }
gfCNCPoint5[2399] = {X 411.5985, Y 79.5924, Z -3.3333, A 0.000, B 0.000, C 0.000 }
gfCNCPoint5[2400] = {X 411.5985, Y 79.5924, Z -6.3333, A 0.000, B 0.000, C 0.000 }
gfCNCPoint5[2401] = {X 413.7988, Y 83.0282, Z -6.3333, A 0.000, B 0.000, C 0.000 }
gfCNCPoint5[2402] = {X 428.0538, Y 73.8996, Z -6.3333, A 0.000, B 0.000, C 0.000 }
gfCNCPoint5[2403] = {X 403.7555, Y 64.3665, Z -6.3333, A 0.000, B 0.000, C 0.000 }
gfCNCPoint5[2404] = {X 402.0595, Y 63.8051, Z -6.3333, A 0.000, B 0.000, C 0.000 }
gfCNCPoint5[2405] = {X 400.3123, Y 63.4328, Z -6.3333, A 0.000, B 0.000, C 0.000 }
gfCNCPoint5[2406] = {X 398.5347, Y 63.2540, Z -6.3333, A 0.000, B 0.000, C 0.000 }
gfCNCPoint5[2407] = {X 397.5822, Y 63.1425, Z -6.3333, A 0.000, B 0.000, C 0.000 }
gfCNCPoint5[2408] = {X 396.6778, Y 62.8236, Z -6.3333, A 0.000, B 0.000, C 0.000 }
gfCNCPoint5[2409] = {X 395.8660, Y 62.3130, Z -6.3333, A 0.000, B 0.000, C 0.000 }
gfCNCPoint5[2410] = {X 395.1869, Y 61.6359, Z -6.3333, A 0.000, B 0.000, C 0.000 }
gfCNCPoint5[2411] = {X 394.6738, Y 60.8256, Z -6.3333, A 0.000, B 0.000, C 0.000 }
gfCNCPoint5[2412] = {X 394.3522, Y 59.9221, Z -6.3333, A 0.000, B 0.000, C 0.000 }
gfCNCPoint5[2413] = {X 394.2379, Y 58.9699, Z -6.3333, A 0.000, B 0.000, C 0.000 }
gfCNCPoint5[2414] = {X 394.2377, Y 58.0000, Z -6.3333, A 0.000, B 0.000, C 0.000 }
gfCNCPoint5[2415] = {X 394.3460, Y 57.0387, Z -6.3333, A 0.000, B 0.000, C 0.000 }
gfCNCPoint5[2416] = {X 394.6655, Y 56.1256, Z -6.3333, A 0.000, B 0.000, C 0.000 }
gfCNCPoint5[2417] = {X 395.1802, Y 55.3065, Z -6.3333, A 0.000, B 0.000, C 0.000 }
gfCNCPoint5[2418] = {X 395.8642, Y 54.6225, Z -6.3333, A 0.000, B 0.000, C 0.000 }
gfCNCPoint5[2419] = {X 396.6833, Y 54.1078, Z -6.3333, A 0.000, B 0.000, C 0.000 }
gfCNCPoint5[2420] = {X 397.5964, Y 53.7883, Z -6.3333, A 0.000, B 0.000, C 0.000 }
gfCNCPoint5[2421] = {X 398.5577, Y 53.6800, Z -6.3333, A 0.000, B 0.000, C 0.000 }
gfCNCPoint5[2422] = {X 419.4886, Y 53.6800, Z -6.3333, A 0.000, B 0.000, C 0.000 }
gfCNCPoint5[2423] = {X 420.4499, Y 53.7883, Z -6.3333, A 0.000, B 0.000, C 0.000 }
